% RSLogix 500 project sdss.RSS %
PROJECT "SDSS"    % processor: SLC 500, 1747-L542 %

PROGRAM FILES
  LAD 2 "MAIN"  21 rungs  %  Main Ladder Logic Program File %
  LAD 3 "TEL AZ"  17 rungs  % Telescope Azimuth Motion Control Logic File %
  LAD 5 "TEL ALT"  28 rungs  % telescope Axis Motion Control Logic File %
  LAD 7 "TEL ROT"  7 rungs  % Telescope Rotator Axis Motion Control Logic File %
  LAD 8 "INST LIFT"  106 rungs  % Instrument Lift Motion Control Logic File %
  LAD 9 "INST LATCH"  114 rungs  % Instrument Latch Control Box File %
  LAD 10 "DATA TRANS"  3 rungs  % Data Transfer subroutine for DH+ link to VME %
  LAD 11 "BRAKE STOP"  13 rungs
  LAD 12 "E-STOP SW"  19 rungs
  LAD 13 "SPEC CONT"  14 rungs  % Spectrograph Controls %
  LAD 14 "FLAT FIELD"  17 rungs  % Flat Field Lamp Controls %
  LAD 15 "FLEXANALOG"  8 rungs  % Flex I/O Analog Routines %

DATA FILES
  O0   92 elements
  I1   98 elements
  S2   164 elements
  B3   109 elements
  T4   19 elements
  C5   1 elements
  R6   1 elements
  N7   74 elements
  F8   105 elements
  B9   256 elements
  B10   48 elements
  B11   1 elements
  F12   20 elements
  B13 B13  1 elements
  N14 N14  50 elements

LADDER 2 "MAIN"    %  Main Ladder Logic Program File %
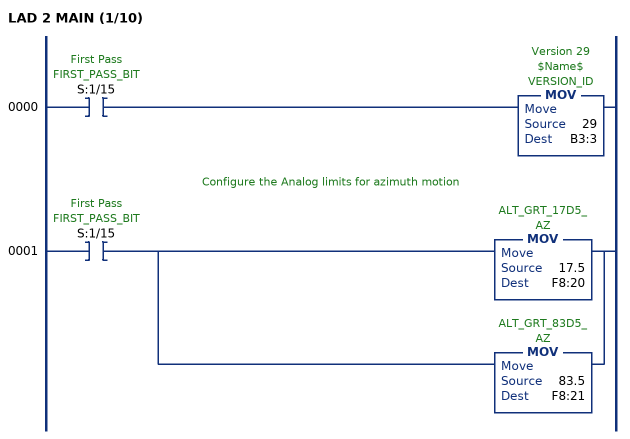
% Rung: 0 %
SOR XIC S:1/15 MOV 29 B3:3 EOR
%   S:1/15  FIRST_PASS_BIT  "First Pass" %
%   B3:3  VERSION_ID  "Version 29 $Name$" %
% Rung: 1 %
% Configure the Analog limits for azimuth motion %
SOR XIC S:1/15 BST MOV 17.5 F8:20 NXB MOV 83.5 F8:21 BND EOR
%   S:1/15  FIRST_PASS_BIT  "First Pass" %
%   F8:20  ALT_GRT_17D5_AZ %
%   F8:21  ALT_GRT_83D5_AZ %

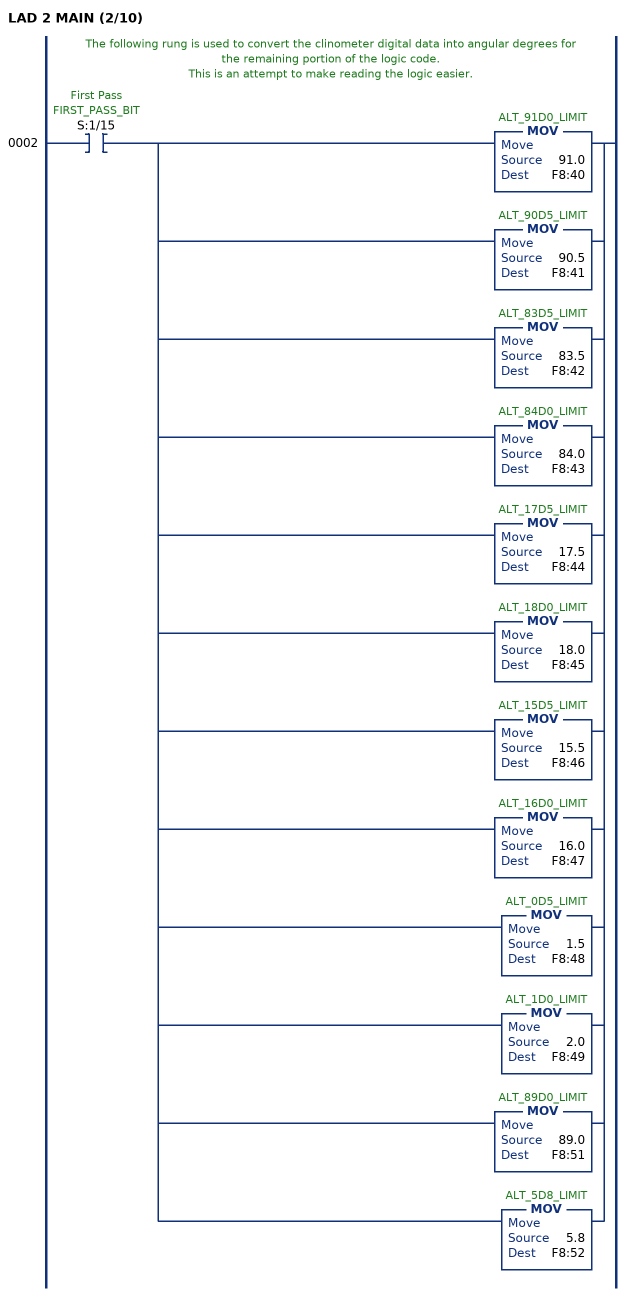
% Rung: 2 %
% The following rung is used to convert the clinometer digital data into angular degrees for the remaining portion of the logic code.
% This is an attempt to make reading the logic easier. %
SOR XIC S:1/15 BST MOV 91.0 F8:40 NXB MOV 90.5 F8:41 NXB MOV 83.5 F8:42 NXB MOV 84.0 F8:43 NXB MOV 17.5 F8:44 NXB MOV 18.0 F8:45 NXB MOV 15.5 F8:46 NXB MOV 16.0 F8:47 NXB MOV 1.5 F8:48 NXB MOV 2.0 F8:49 NXB MOV 89.0 F8:51 NXB MOV 5.8 F8:52 BND EOR
%   S:1/15  FIRST_PASS_BIT  "First Pass" %
%   F8:40  ALT_91D0_LIMIT %
%   F8:41  ALT_90D5_LIMIT %
%   F8:42  ALT_83D5_LIMIT %
%   F8:43  ALT_84D0_LIMIT %
%   F8:44  ALT_17D5_LIMIT %
%   F8:45  ALT_18D0_LIMIT %
%   F8:46  ALT_15D5_LIMIT %
%   F8:47  ALT_16D0_LIMIT %
%   F8:48  ALT_0D5_LIMIT %
%   F8:49  ALT_1D0_LIMIT %
%   F8:51  ALT_89D0_LIMIT %
%   F8:52  ALT_5D8_LIMIT %

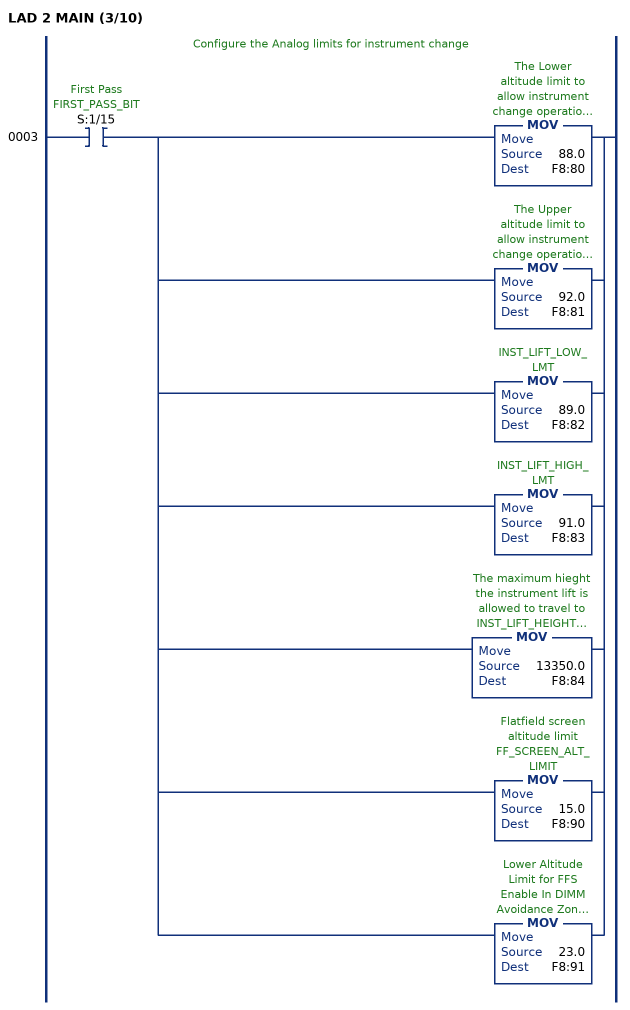
% Rung: 3 %
% Configure the Analog limits for instrument change %
SOR XIC S:1/15 BST MOV 88.0 F8:80 NXB MOV 92.0 F8:81 NXB MOV 89.0 F8:82 NXB MOV 91.0 F8:83 NXB MOV 13350.0 F8:84 NXB BST MOV 15.0 F8:90 NXB MOV 23.0 F8:91 BND BND EOR
%   S:1/15  FIRST_PASS_BIT  "First Pass" %
%   F8:80  INST_CHG_LOW_LMT  "The Lower altitude limit to allow instrument change operations" %
%   F8:81  INST_CHG_HIGH_LMT  "The Upper altitude limit to allow instrument change operations" %
%   F8:82  INST_LIFT_LOW_LMT %
%   F8:83  INST_LIFT_HIGH_LMT %
%   F8:84  INST_LIFT_HEIGHT_MAX  "The maximum hieght the instrument lift is allowed to travel to" %
%   F8:90  FF_SCREEN_ALT_LIMIT  "Flatfield screen altitude limit" %
%   F8:91  FFS_DIMM_ALT_LIM  "Lower Altitude Limit for FFS Enable In DIMM Avoidance Zone" %

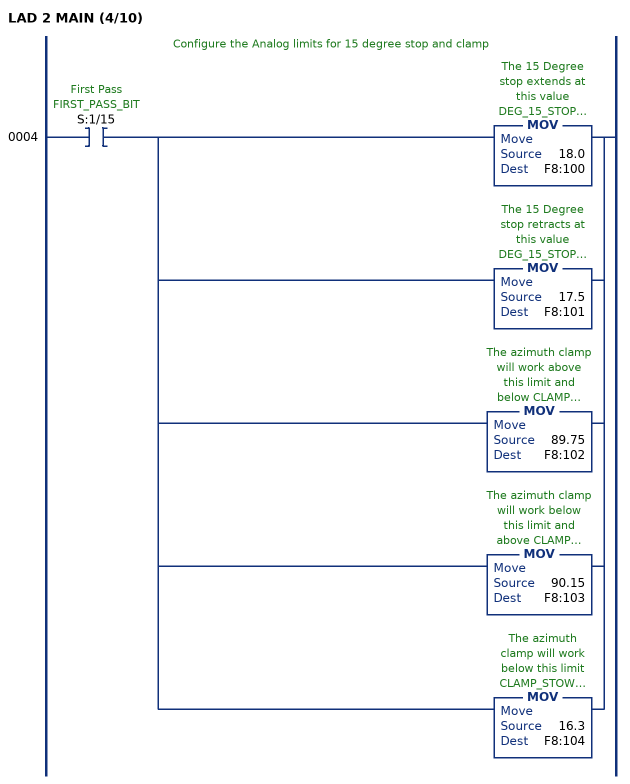
% Rung: 4 %
% Configure the Analog limits for 15 degree stop and clamp %
SOR XIC S:1/15 BST MOV 18.0 F8:100 NXB MOV 17.5 F8:101 NXB MOV 89.75 F8:102 NXB MOV 90.15 F8:103 NXB MOV 16.3 F8:104 BND EOR
%   S:1/15  FIRST_PASS_BIT  "First Pass" %
%   F8:100  DEG_15_STOP_EXT_LMT  "The 15 Degree stop extends at this value" %
%   F8:101  DEG_15_STOP_RET_LMT  "The 15 Degree stop retracts at this value" %
%   F8:102  CLAMP_LOW_LIMIT  "The azimuth clamp will work above this limit and below CLAMP_HIGH_LIMIT" %
%   F8:103  CLAMP_HIGH_LIMIT  "The azimuth clamp will work below this limit and above CLAMP_LOW_LIMIT" %
%   F8:104  CLAMP_STOW_LIMIT  "The azimuth clamp will work below this limit" %

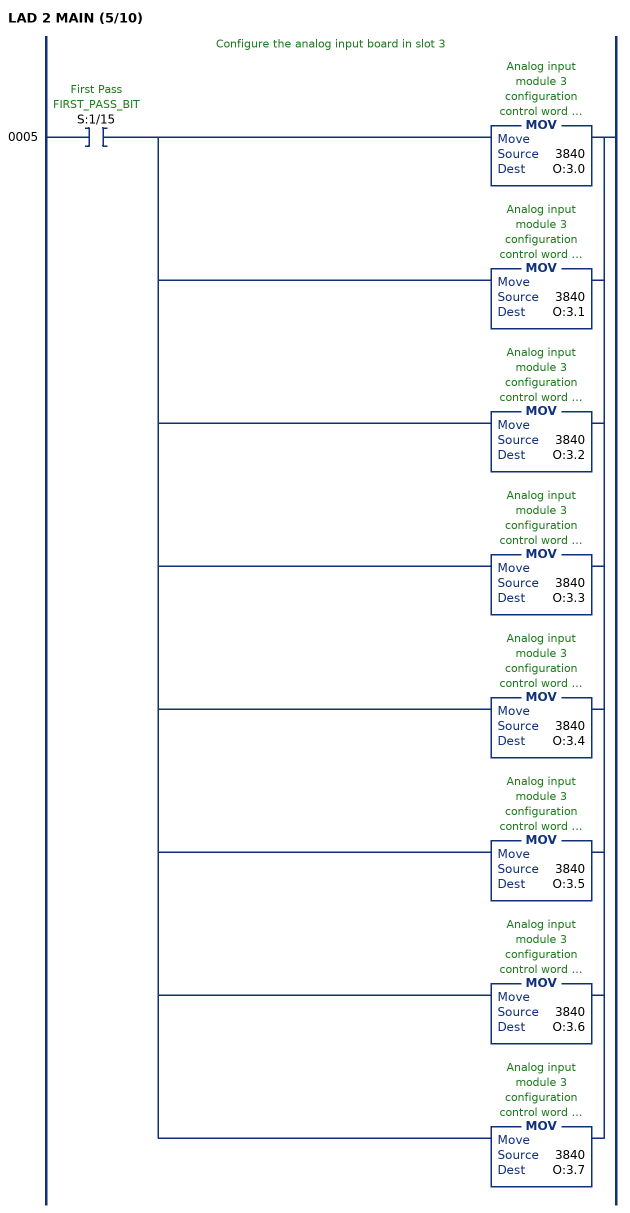
% Rung: 5 %
% Configure the analog input board in slot 3 %
SOR XIC S:1/15 BST MOV 3840 O:3.0 NXB MOV 3840 O:3.1 NXB MOV 3840 O:3.2 NXB MOV 3840 O:3.3 NXB MOV 3840 O:3.4 NXB MOV 3840 O:3.5 NXB MOV 3840 O:3.6 NXB MOV 3840 O:3.7 BND EOR
%   S:1/15  FIRST_PASS_BIT  "First Pass" %
%   O:3.0  AZ_1_VOLTAGE_CONFIG  "Analog input module 3 configuration control word 0" %
%   O:3.1  AZ_1_CURRENT_CONFIG  "Analog input module 3 configuration control word 1" %
%   O:3.2  AZ_2_VOLTAGE_CONFIG  "Analog input module 3 configuration control word 2" %
%   O:3.3  AZ_2_CURRENT_CONFIG  "Analog input module 3 configuration control word 3" %
%   O:3.4  ALT_1_VOLTAGE_CONFIG  "Analog input module 3 configuration control word 4" %
%   O:3.5  ALT_1_CURRENT_CONFIG  "Analog input module 3 configuration control word 5" %
%   O:3.6  ALT_2_VOLTAGE_CONFIG  "Analog input module 3 configuration control word 6" %
%   O:3.7  ALT_2_CURRENT_CONFIG  "Analog input module 3 configuration control word 7" %

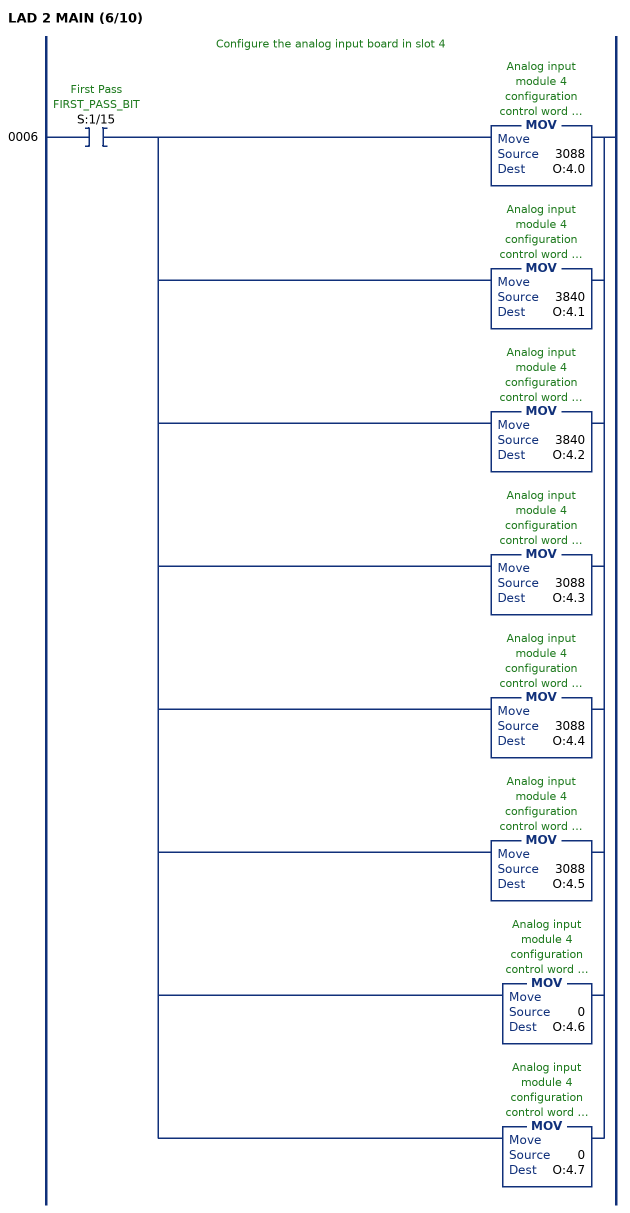
% Rung: 6 %
% Configure the analog input board in slot 4 %
SOR XIC S:1/15 BST MOV 3088 O:4.0 NXB MOV 3840 O:4.1 NXB MOV 3840 O:4.2 NXB MOV 3088 O:4.3 NXB MOV 3088 O:4.4 NXB MOV 3088 O:4.5 NXB MOV 0 O:4.6 NXB MOV 0 O:4.7 BND EOR
%   S:1/15  FIRST_PASS_BIT  "First Pass" %
%   O:4.0  ALT_POSITION_CONFIG  "Analog input module 4 configuration control word 0" %
%   O:4.1  ROT_1_VOLTAGE_CONFIG  "Analog input module 4 configuration control word 1" %
%   O:4.2  ROT_1_CURRENT_CONFIG  "Analog input module 4 configuration control word 2" %
%   O:4.3  UMBILICAL_DIST_CONFI  "Analog input module 4 configuration control word 3" %
%   O:4.4  INST_LIFT_FORCE_CONF  "Analog input module 4 configuration control word 4" %
%   O:4.5  INST_LIFT_DIST_CONFI  "Analog input module 4 configuration control word 5" %
%   O:4.6  I_4_ANALOG_6_CONFIG  "Analog input module 4 configuration control word 6" %
%   O:4.7  I_4_ANALOG_7_CONFIG  "Analog input module 4 configuration control word 7" %

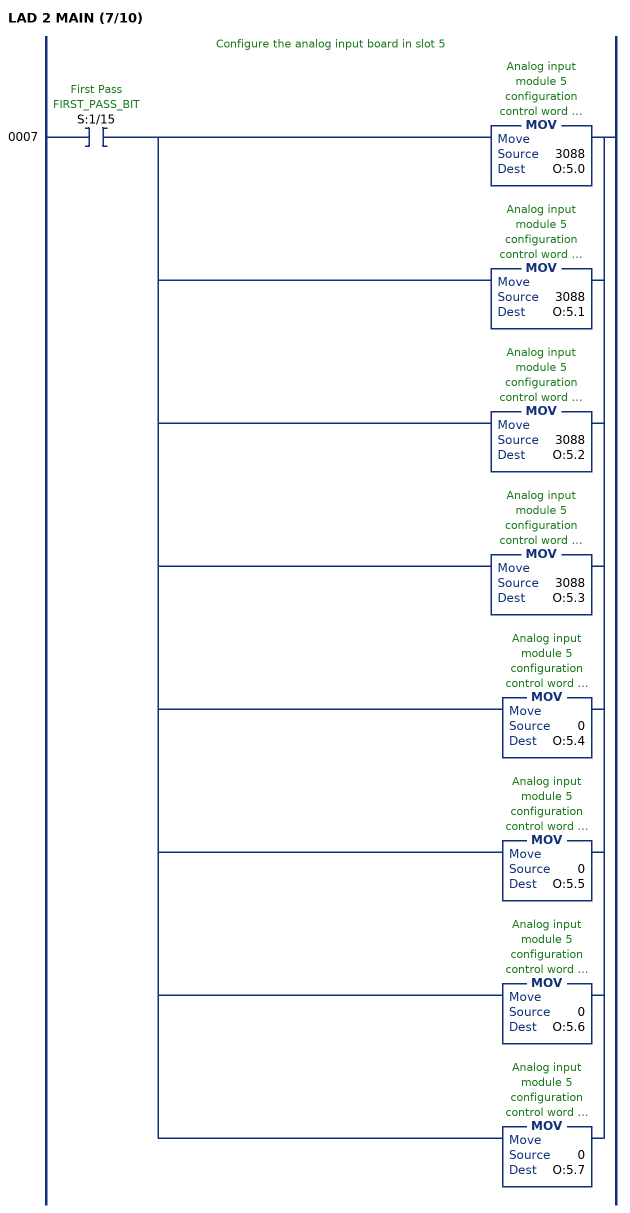
% Rung: 7 %
% Configure the analog input board in slot 5 %
SOR XIC S:1/15 BST MOV 3088 O:5.0 NXB MOV 3088 O:5.1 NXB MOV 3088 O:5.2 NXB MOV 3088 O:5.3 NXB MOV 0 O:5.4 NXB MOV 0 O:5.5 NXB MOV 0 O:5.6 NXB MOV 0 O:5.7 BND EOR
%   S:1/15  FIRST_PASS_BIT  "First Pass" %
%   O:5.0  CNTRWHT_1_POS_CONFIG  "Analog input module 5 configuration control word 0" %
%   O:5.1  CNTRWHT_2_POS_CONFIG  "Analog input module 5 configuration control word 1" %
%   O:5.2  CNTRWHT_3_POS_CONFIG  "Analog input module 5 configuration control word 2" %
%   O:5.3  CNTRWHT_4_POS_CONFIG  "Analog input module 5 configuration control word 3" %
%   O:5.4  I_5_ANALOG_4_CONFIG  "Analog input module 5 configuration control word 4" %
%   O:5.5  I_5_ANALOG_5_CONFIG  "Analog input module 5 configuration control word 5" %
%   O:5.6  I_5_ANALOG_6_CONFIG  "Analog input module 5 configuration control word 6" %
%   O:5.7  I_5_ANALOG_7_CONFIG  "Analog input module 5 configuration control word 7" %

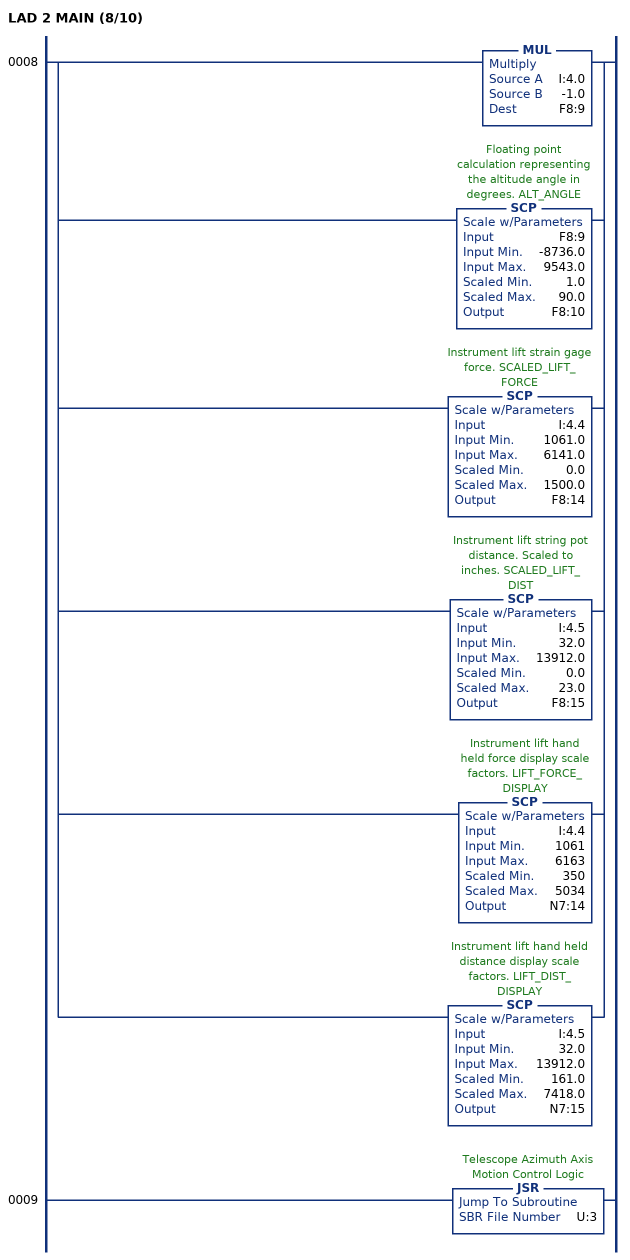
% Rung: 8 %
SOR BST MUL I:4.0 -1.0 F8:9 NXB SCP F8:9 -8736.0 9543.0 1.0 90.0 F8:10 NXB SCP I:4.4 1061.0 6141.0 0.0 1500.0 F8:14 NXB SCP I:4.5 32.0 13912.0 0.0 23.0 F8:15 NXB SCP I:4.4 1061 6163 350 5034 N7:14 NXB SCP I:4.5 32.0 13912.0 161.0 7418.0 N7:15 BND EOR
%   I:4.0  ALT_POSITION  "Altitude clinometer raw position value." %
%   F8:10  ALT_ANGLE  "Floating point calculation representing the altitude angle in degrees." %
%   I:4.4  INST_LIFT_FORCE  "Instrument lift strain gauge value." %
%   F8:14  SCALED_LIFT_FORCE  "Instrument lift strain gage force." %
%   I:4.5  INST_LIFT_DIST  "Instrument lift string pot distance value. Scale = .001,per count." 0" %
%   F8:15  SCALED_LIFT_DIST  "Instrument lift string pot distance. Scaled to inches." %
%   N7:14  LIFT_FORCE_DISPLAY  "Instrument lift hand held force display scale factors." %
%   N7:15  LIFT_DIST_DISPLAY  "Instrument lift hand held distance display scale factors." %
% Rung: 9 %
SOR JSR U:3 EOR
%   U:3  "Telescope Azimuth Axis Motion Control Logic" %

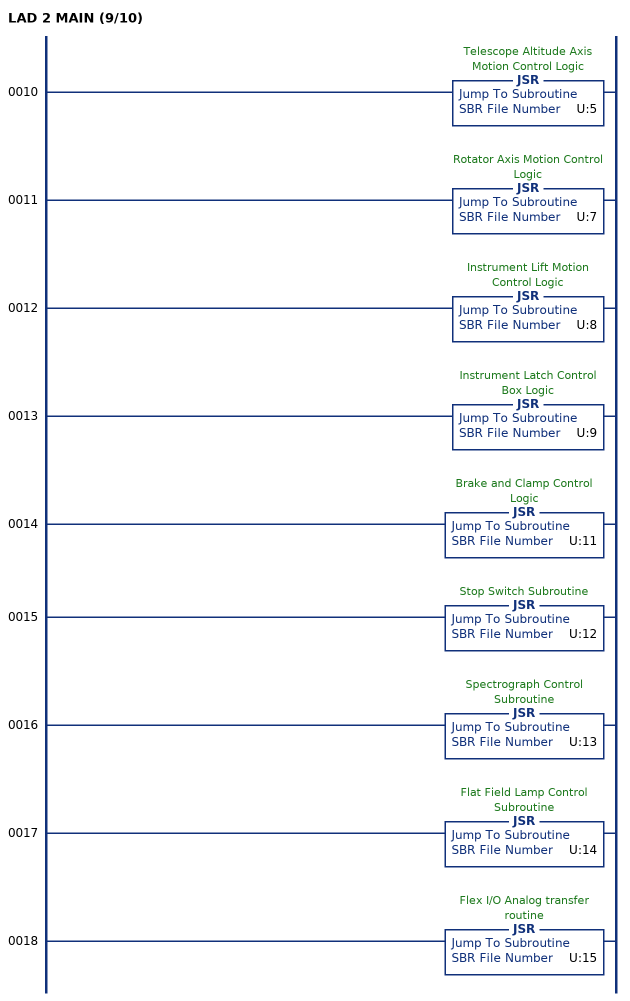
% Rung: 10 %
SOR JSR U:5 EOR
%   U:5  "Telescope Altitude Axis Motion Control Logic" %
% Rung: 11 %
SOR JSR U:7 EOR
%   U:7  "Rotator Axis Motion Control Logic" %
% Rung: 12 %
SOR JSR U:8 EOR
%   U:8  "Instrument Lift Motion Control Logic" %
% Rung: 13 %
SOR JSR U:9 EOR
%   U:9  "Instrument Latch Control Box Logic" %
% Rung: 14 %
SOR JSR U:11 EOR
%   U:11  "Brake and Clamp Control Logic" %
% Rung: 15 %
SOR JSR U:12 EOR
%   U:12  "Stop Switch Subroutine" %
% Rung: 16 %
SOR JSR U:13 EOR
%   U:13  "Spectrograph Control Subroutine" %
% Rung: 17 %
SOR JSR U:14 EOR
%   U:14  "Flat Field Lamp Control Subroutine" %
% Rung: 18 %
SOR JSR U:15 EOR
%   U:15  "Flex I/O Analog transfer routine" %

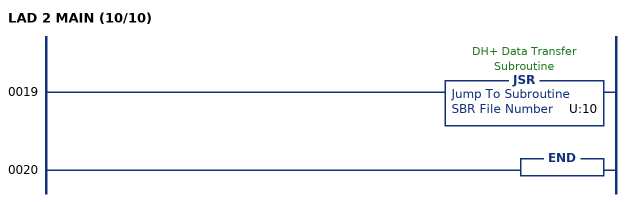
% Rung: 19 %
SOR JSR U:10 EOR
%   U:10  "DH+ Data Transfer Subroutine" %
% Rung: 20 %
SOR END EOR

LADDER 3 "TEL AZ"    % Telescope Azimuth Motion Control Logic File %
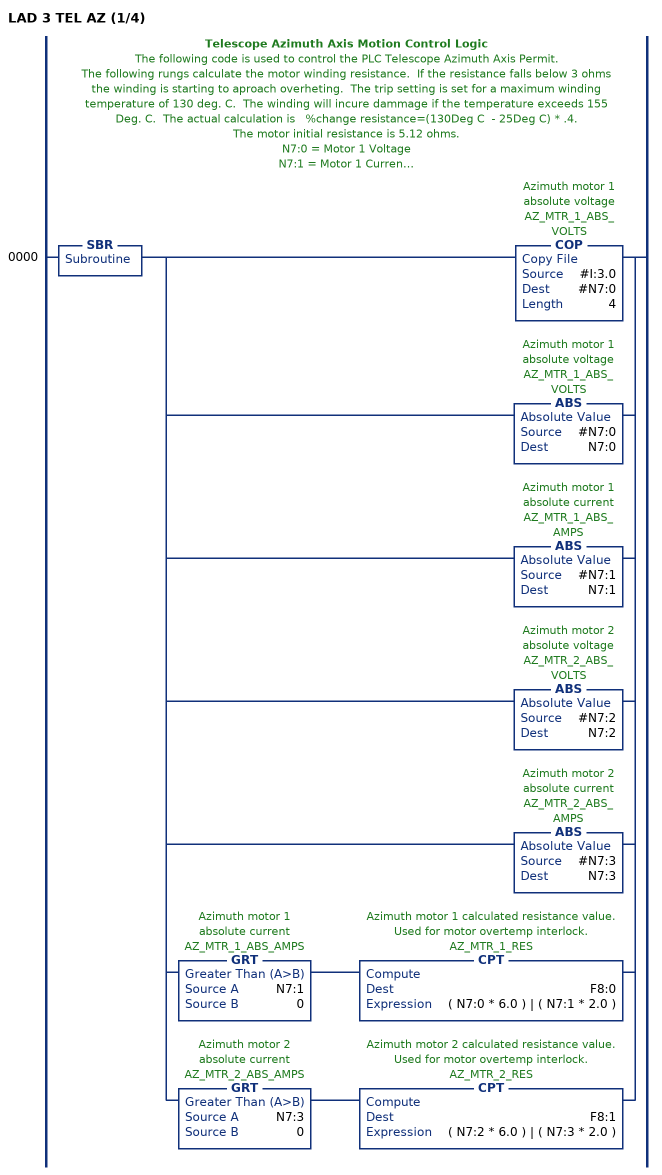
% Rung: 0 %
% TITLE: Telescope Azimuth Axis Motion Control Logic %
% The following code is used to control the PLC Telescope Azimuth Axis Permit.
% 
% 
% The following rungs calculate the motor winding resistance.  If the resistance falls below 3 ohms the winding is starting to aproach overheting.  The trip setting is set for a maximum winding temperature of 130 deg. C.  The winding will incure dammage if the temperature exceeds 155 Deg. C.  The actual calculation is   %change resistance=(130Deg C  - 25Deg C) * .4.
% 
% The motor initial resistance is 5.12 ohms.
% 
% 
% N7:0 = Motor 1 Voltage
% N7:1 = Motor 1 Current
% N7:2 = Motor 2 Voltage
% N7:3 = Motor 2 Current
% 
% If the voltage and current are not above 500 counts, then the resistance calculation is considdered invalid and an output permit is provided. %
SOR SBR BST COP #I:3.0 #N7:0 4 NXB ABS #N7:0 N7:0 NXB ABS #N7:1 N7:1 NXB ABS #N7:2 N7:2 NXB ABS #N7:3 N7:3 NXB GRT N7:1 0 CPT F8:0 " ( N7:0 * 6.0 ) | ( N7:1 * 2.0 ) " NXB GRT N7:3 0 CPT F8:1 " ( N7:2 * 6.0 ) | ( N7:3 * 2.0 ) " BND EOR
%   I:3.0  AZ_1_VOLTAGE  "Azimuth motor 1 voltage." %
%   N7:0  AZ_MTR_1_ABS_VOLTS  "Azimuth motor 1 absolute voltage" %
%   N7:1  AZ_MTR_1_ABS_AMPS  "Azimuth motor 1 absolute current" %
%   N7:2  AZ_MTR_2_ABS_VOLTS  "Azimuth motor 2 absolute voltage" %
%   N7:3  AZ_MTR_2_ABS_AMPS  "Azimuth motor 2 absolute current" %
%   F8:0  AZ_MTR_1_RES  "Azimuth motor 1 calculated resistance value. Used for motor overtemp interlock." %
%   F8:1  AZ_MTR_2_RES  "Azimuth motor 2 calculated resistance value. Used for motor overtemp interlock." %

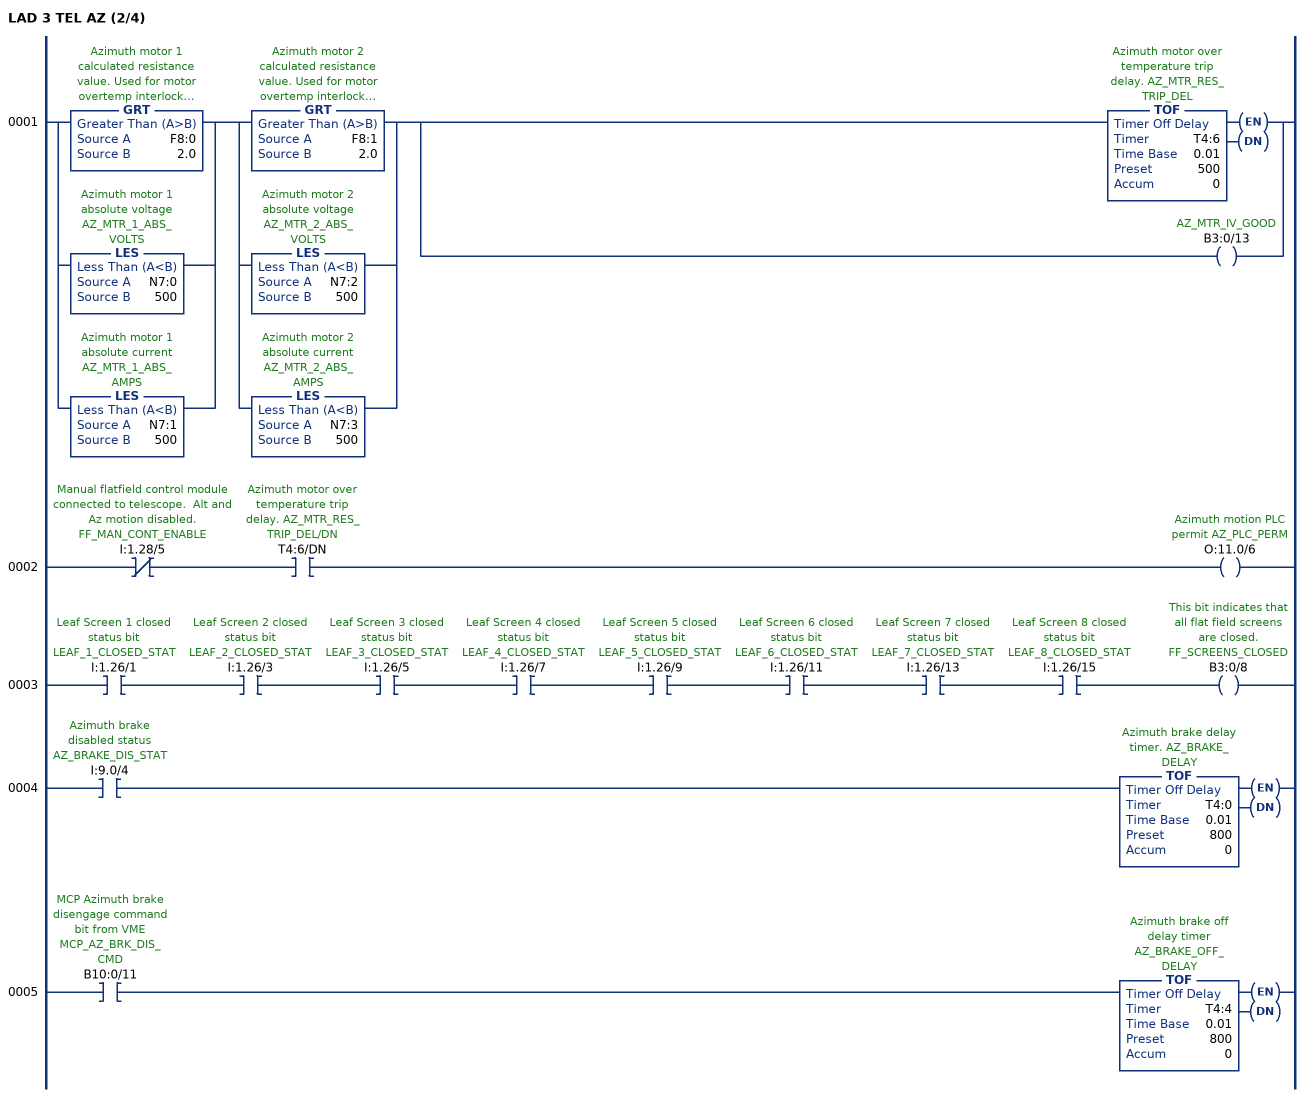
% Rung: 1 %
SOR BST GRT F8:0 2.0 NXB LES N7:0 500 NXB LES N7:1 500 BND BST GRT F8:1 2.0 NXB LES N7:2 500 NXB LES N7:3 500 BND BST TOF T4:6 0.01 500 0 NXB OTE B3:0/13 BND EOR
%   F8:0  AZ_MTR_1_RES  "Azimuth motor 1 calculated resistance value. Used for motor overtemp interlock." %
%   N7:0  AZ_MTR_1_ABS_VOLTS  "Azimuth motor 1 absolute voltage" %
%   N7:1  AZ_MTR_1_ABS_AMPS  "Azimuth motor 1 absolute current" %
%   F8:1  AZ_MTR_2_RES  "Azimuth motor 2 calculated resistance value. Used for motor overtemp interlock." %
%   N7:2  AZ_MTR_2_ABS_VOLTS  "Azimuth motor 2 absolute voltage" %
%   N7:3  AZ_MTR_2_ABS_AMPS  "Azimuth motor 2 absolute current" %
%   T4:6  AZ_MTR_RES_TRIP_DEL  "Azimuth motor over temperature trip delay." %
%   B3:0/13  AZ_MTR_IV_GOOD %
% Rung: 2 %
SOR XIO I:1.28/5 XIC T4:6/DN OTE O:11.0/6 EOR
%   I:1.28/5  FF_MAN_CONT_ENABLE  "Manual flatfield control module connected to telescope.  Alt and Az motion disabled." %
%   T4:6  AZ_MTR_RES_TRIP_DEL  "Azimuth motor over temperature trip delay." %
%   O:11.0/6  AZ_PLC_PERM  "Azimuth motion PLC permit" %
% Rung: 3 %
SOR XIC I:1.26/1 XIC I:1.26/3 XIC I:1.26/5 XIC I:1.26/7 XIC I:1.26/9 XIC I:1.26/11 XIC I:1.26/13 XIC I:1.26/15 OTE B3:0/8 EOR
%   I:1.26/1  LEAF_1_CLOSED_STAT  "Leaf Screen 1 closed status bit" %
%   I:1.26/3  LEAF_2_CLOSED_STAT  "Leaf Screen 2 closed status bit" %
%   I:1.26/5  LEAF_3_CLOSED_STAT  "Leaf Screen 3 closed status bit" %
%   I:1.26/7  LEAF_4_CLOSED_STAT  "Leaf Screen 4 closed status bit" %
%   I:1.26/9  LEAF_5_CLOSED_STAT  "Leaf Screen 5 closed status bit" %
%   I:1.26/11  LEAF_6_CLOSED_STAT  "Leaf Screen 6 closed status bit" %
%   I:1.26/13  LEAF_7_CLOSED_STAT  "Leaf Screen 7 closed status bit" %
%   I:1.26/15  LEAF_8_CLOSED_STAT  "Leaf Screen 8 closed status bit" %
%   B3:0/8  FF_SCREENS_CLOSED  "This bit indicates that all flat field screens are closed." %
% Rung: 4 %
SOR XIC I:9.0/4 TOF T4:0 0.01 800 0 EOR
%   I:9.0/4  AZ_BRAKE_DIS_STAT  "Azimuth brake disabled status" %
%   T4:0  AZ_BRAKE_DELAY  "Azimuth brake delay timer." %
% Rung: 5 %
SOR XIC B10:0/11 TOF T4:4 0.01 800 0 EOR
%   B10:0/11  MCP_AZ_BRK_DIS_CMD  "MCP Azimuth brake disengage command bit from VME" %
%   T4:4  AZ_BRAKE_OFF_DELAY  "Azimuth brake off delay timer" %

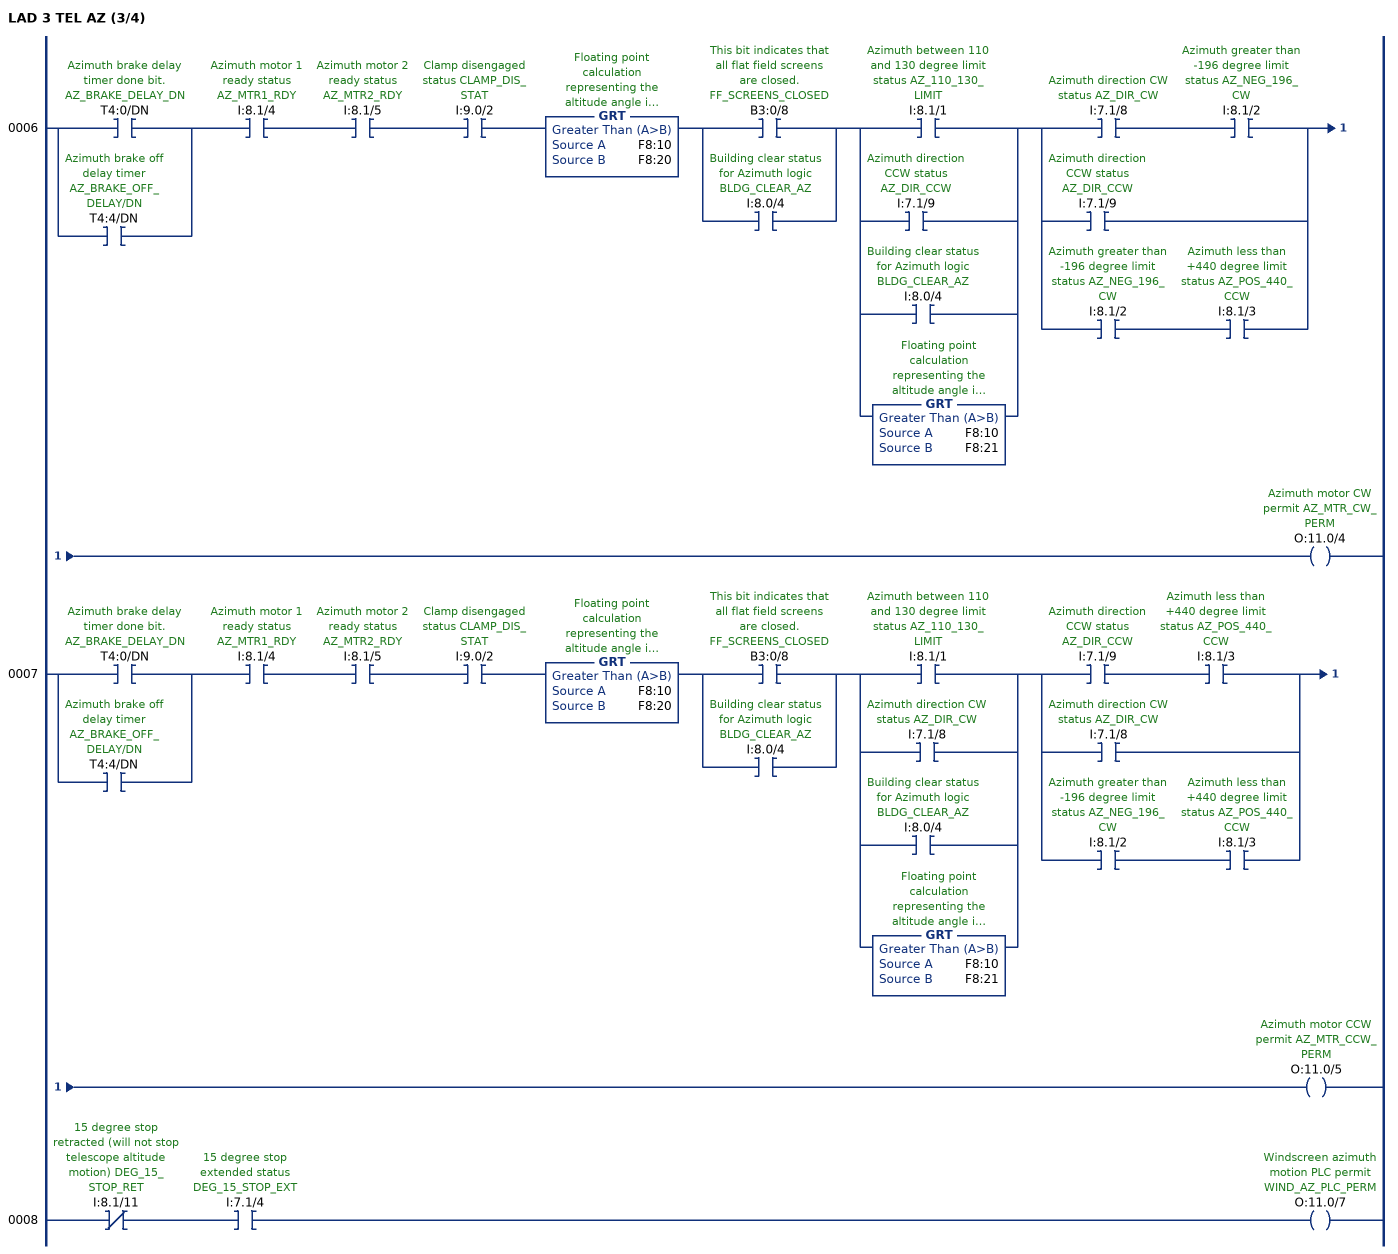
% Rung: 6 %
SOR BST XIC T4:0/DN NXB XIC T4:4/DN BND XIC I:8.1/4 XIC I:8.1/5 XIC I:9.0/2 GRT F8:10 F8:20 BST XIC B3:0/8 NXB XIC I:8.0/4 BND BST XIC I:8.1/1 NXB XIC I:7.1/9 NXB XIC I:8.0/4 NXB GRT F8:10 F8:21 BND BST XIC I:7.1/8 XIC I:8.1/2 NXB XIC I:7.1/9 NXB XIC I:8.1/2 XIC I:8.1/3 BND OTE O:11.0/4 EOR
%   T4:0/DN  AZ_BRAKE_DELAY_DN  "Azimuth brake delay timer done bit." %
%   T4:4  AZ_BRAKE_OFF_DELAY  "Azimuth brake off delay timer" %
%   I:8.1/4  AZ_MTR1_RDY  "Azimuth motor 1 ready status" %
%   I:8.1/5  AZ_MTR2_RDY  "Azimuth motor 2 ready status" %
%   I:9.0/2  CLAMP_DIS_STAT  "Clamp disengaged status" %
%   F8:10  ALT_ANGLE  "Floating point calculation representing the altitude angle in degrees." %
%   F8:20  ALT_GRT_17D5_AZ %
%   B3:0/8  FF_SCREENS_CLOSED  "This bit indicates that all flat field screens are closed." %
%   I:8.0/4  BLDG_CLEAR_AZ  "Building clear status for Azimuth logic" %
%   I:8.1/1  AZ_110_130_LIMIT  "Azimuth between 110 and 130 degree limit status" %
%   I:7.1/9  AZ_DIR_CCW  "Azimuth direction CCW status" %
%   F8:21  ALT_GRT_83D5_AZ %
%   I:7.1/8  AZ_DIR_CW  "Azimuth direction CW status" %
%   I:8.1/2  AZ_NEG_196_CW  "Azimuth greater than -196 degree limit status" %
%   I:8.1/3  AZ_POS_440_CCW  "Azimuth less than +440 degree limit status" %
%   O:11.0/4  AZ_MTR_CW_PERM  "Azimuth motor CW permit" %
% Rung: 7 %
SOR BST XIC T4:0/DN NXB XIC T4:4/DN BND XIC I:8.1/4 XIC I:8.1/5 XIC I:9.0/2 GRT F8:10 F8:20 BST XIC B3:0/8 NXB XIC I:8.0/4 BND BST XIC I:8.1/1 NXB XIC I:7.1/8 NXB XIC I:8.0/4 NXB GRT F8:10 F8:21 BND BST XIC I:7.1/9 XIC I:8.1/3 NXB XIC I:7.1/8 NXB XIC I:8.1/2 XIC I:8.1/3 BND OTE O:11.0/5 EOR
%   T4:0/DN  AZ_BRAKE_DELAY_DN  "Azimuth brake delay timer done bit." %
%   T4:4  AZ_BRAKE_OFF_DELAY  "Azimuth brake off delay timer" %
%   I:8.1/4  AZ_MTR1_RDY  "Azimuth motor 1 ready status" %
%   I:8.1/5  AZ_MTR2_RDY  "Azimuth motor 2 ready status" %
%   I:9.0/2  CLAMP_DIS_STAT  "Clamp disengaged status" %
%   F8:10  ALT_ANGLE  "Floating point calculation representing the altitude angle in degrees." %
%   F8:20  ALT_GRT_17D5_AZ %
%   B3:0/8  FF_SCREENS_CLOSED  "This bit indicates that all flat field screens are closed." %
%   I:8.0/4  BLDG_CLEAR_AZ  "Building clear status for Azimuth logic" %
%   I:8.1/1  AZ_110_130_LIMIT  "Azimuth between 110 and 130 degree limit status" %
%   I:7.1/8  AZ_DIR_CW  "Azimuth direction CW status" %
%   F8:21  ALT_GRT_83D5_AZ %
%   I:7.1/9  AZ_DIR_CCW  "Azimuth direction CCW status" %
%   I:8.1/3  AZ_POS_440_CCW  "Azimuth less than +440 degree limit status" %
%   I:8.1/2  AZ_NEG_196_CW  "Azimuth greater than -196 degree limit status" %
%   O:11.0/5  AZ_MTR_CCW_PERM  "Azimuth motor CCW permit" %
% Rung: 8 %
SOR XIO I:8.1/11 XIC I:7.1/4 OTE O:11.0/7 EOR
%   I:8.1/11  DEG_15_STOP_RET  "15 degree stop retracted (will not stop telescope altitude motion)" %
%   I:7.1/4  DEG_15_STOP_EXT  "15 degree stop extended status" %
%   O:11.0/7  WIND_AZ_PLC_PERM  "Windscreen azimuth motion PLC permit" %

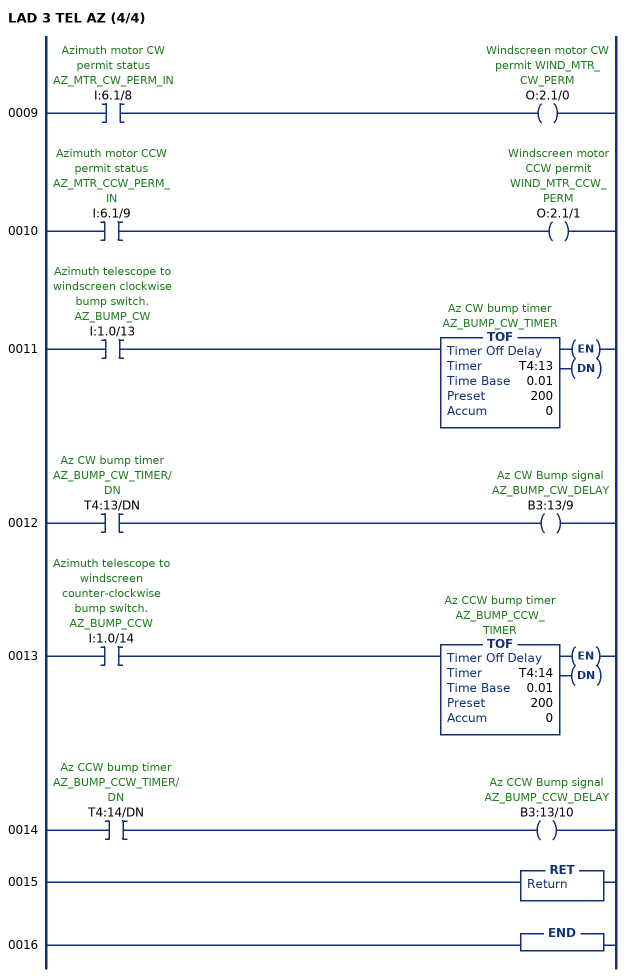
% Rung: 9 %
SOR XIC I:6.1/8 OTE O:2.1/0 EOR
%   I:6.1/8  AZ_MTR_CW_PERM_IN  "Azimuth motor CW permit status" %
%   O:2.1/0  WIND_MTR_CW_PERM  "Windscreen motor CW permit" %
% Rung: 10 %
SOR XIC I:6.1/9 OTE O:2.1/1 EOR
%   I:6.1/9  AZ_MTR_CCW_PERM_IN  "Azimuth motor CCW permit status" %
%   O:2.1/1  WIND_MTR_CCW_PERM  "Windscreen motor CCW permit" %
% Rung: 11 %
SOR XIC I:1.0/13 TOF T4:13 0.01 200 0 EOR
%   I:1.0/13  AZ_BUMP_CW  "Azimuth telescope to windscreen clockwise bump switch." %
%   T4:13  AZ_BUMP_CW_TIMER  "Az CW bump timer" %
% Rung: 12 %
SOR XIC T4:13/DN OTE B3:13/9 EOR
%   T4:13  AZ_BUMP_CW_TIMER  "Az CW bump timer" %
%   B3:13/9  AZ_BUMP_CW_DELAY  "Az CW Bump signal" %
% Rung: 13 %
SOR XIC I:1.0/14 TOF T4:14 0.01 200 0 EOR
%   I:1.0/14  AZ_BUMP_CCW  "Azimuth telescope to windscreen counter-clockwise bump switch." %
%   T4:14  AZ_BUMP_CCW_TIMER  "Az CCW bump timer" %
% Rung: 14 %
SOR XIC T4:14/DN OTE B3:13/10 EOR
%   T4:14  AZ_BUMP_CCW_TIMER  "Az CCW bump timer" %
%   B3:13/10  AZ_BUMP_CCW_DELAY  "Az CCW Bump signal" %
% Rung: 15 %
SOR RET EOR
% Rung: 16 %
SOR END EOR

LADDER 5 "TEL ALT"    % telescope Axis Motion Control Logic File %
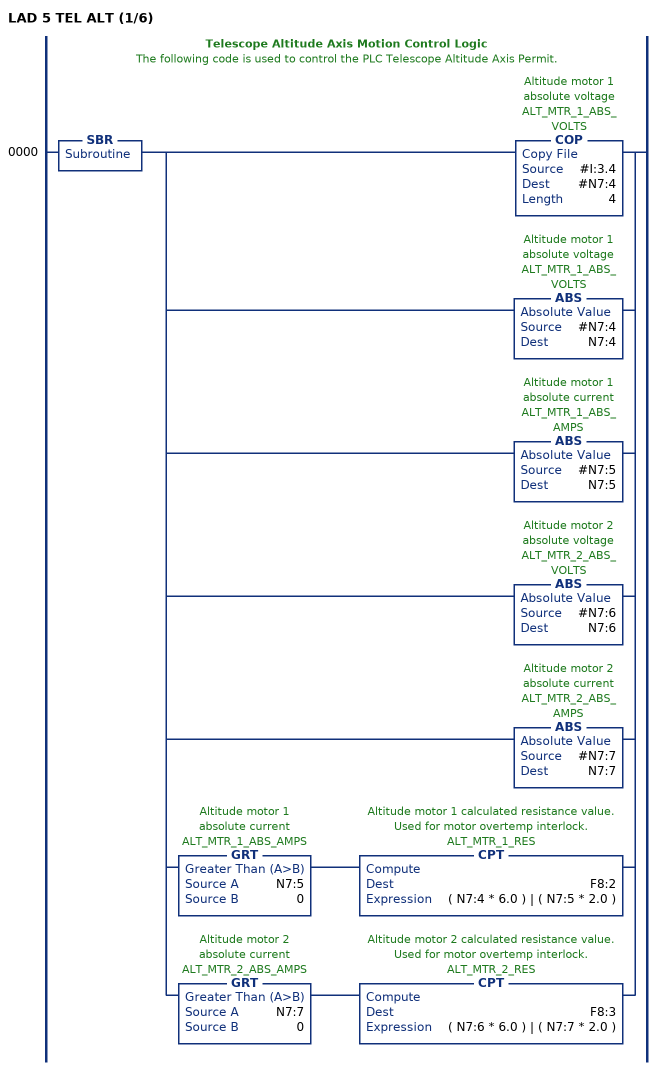
% Rung: 0 %
% TITLE: Telescope Altitude Axis Motion Control Logic %
% The following code is used to control the PLC Telescope Altitude Axis Permit. %
SOR SBR BST COP #I:3.4 #N7:4 4 NXB ABS #N7:4 N7:4 NXB ABS #N7:5 N7:5 NXB ABS #N7:6 N7:6 NXB ABS #N7:7 N7:7 NXB GRT N7:5 0 CPT F8:2 " ( N7:4 * 6.0 ) | ( N7:5 * 2.0 ) " NXB GRT N7:7 0 CPT F8:3 " ( N7:6 * 6.0 ) | ( N7:7 * 2.0 ) " BND EOR
%   I:3.4  ALT_1_VOLTAGE  "Altitude motor 1 voltage." %
%   N7:4  ALT_MTR_1_ABS_VOLTS  "Altitude motor 1 absolute voltage" %
%   N7:5  ALT_MTR_1_ABS_AMPS  "Altitude motor 1 absolute current" %
%   N7:6  ALT_MTR_2_ABS_VOLTS  "Altitude motor 2 absolute voltage" %
%   N7:7  ALT_MTR_2_ABS_AMPS  "Altitude motor 2 absolute current" %
%   F8:2  ALT_MTR_1_RES  "Altitude motor 1 calculated resistance value. Used for motor overtemp interlock." %
%   F8:3  ALT_MTR_2_RES  "Altitude motor 2 calculated resistance value. Used for motor overtemp interlock." %

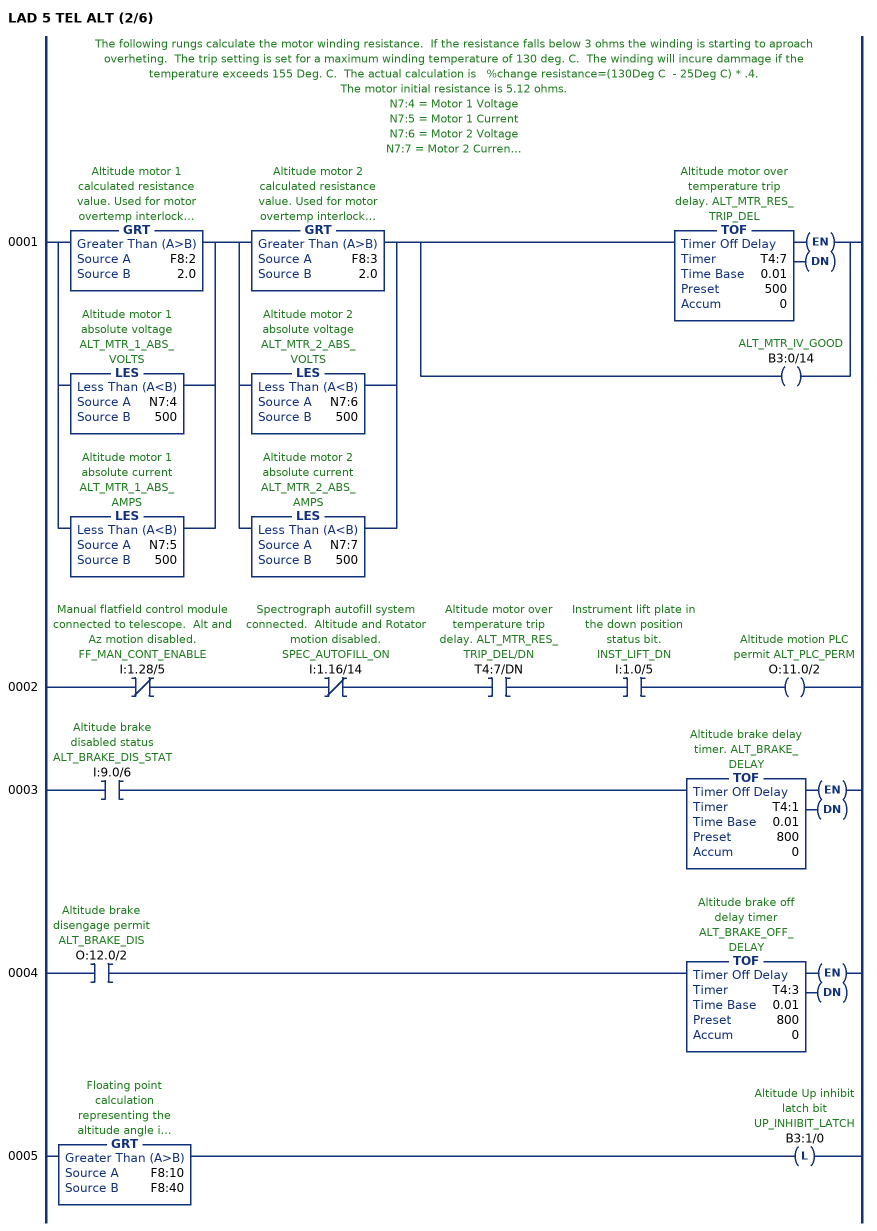
% Rung: 1 %
% The following rungs calculate the motor winding resistance.  If the resistance falls below 3 ohms the winding is starting to aproach overheting.  The trip setting is set for a maximum winding temperature of 130 deg. C.  The winding will incure dammage if the temperature exceeds 155 Deg. C.  The actual calculation is   %change resistance=(130Deg C  - 25Deg C) * .4.
% 
% The motor initial resistance is 5.12 ohms.
% 
% 
% 
% N7:4 = Motor 1 Voltage
% N7:5 = Motor 1 Current
% N7:6 = Motor 2 Voltage
% N7:7 = Motor 2 Current
% 
% If the voltage and current are not above 500 counts, then the resistance calculation is considdered invalid and an output permit is provided. %
SOR BST GRT F8:2 2.0 NXB LES N7:4 500 NXB LES N7:5 500 BND BST GRT F8:3 2.0 NXB LES N7:6 500 NXB LES N7:7 500 BND BST TOF T4:7 0.01 500 0 NXB OTE B3:0/14 BND EOR
%   F8:2  ALT_MTR_1_RES  "Altitude motor 1 calculated resistance value. Used for motor overtemp interlock." %
%   N7:4  ALT_MTR_1_ABS_VOLTS  "Altitude motor 1 absolute voltage" %
%   N7:5  ALT_MTR_1_ABS_AMPS  "Altitude motor 1 absolute current" %
%   F8:3  ALT_MTR_2_RES  "Altitude motor 2 calculated resistance value. Used for motor overtemp interlock." %
%   N7:6  ALT_MTR_2_ABS_VOLTS  "Altitude motor 2 absolute voltage" %
%   N7:7  ALT_MTR_2_ABS_AMPS  "Altitude motor 2 absolute current" %
%   T4:7  ALT_MTR_RES_TRIP_DEL  "Altitude motor over temperature trip delay." %
%   B3:0/14  ALT_MTR_IV_GOOD %
% Rung: 2 %
SOR XIO I:1.28/5 XIO I:1.16/14 XIC T4:7/DN XIC I:1.0/5 OTE O:11.0/2 EOR
%   I:1.28/5  FF_MAN_CONT_ENABLE  "Manual flatfield control module connected to telescope.  Alt and Az motion disabled." %
%   I:1.16/14  SPEC_AUTOFILL_ON  "Spectrograph autofill system connected.  Altitude and Rotator motion disabled." %
%   T4:7  ALT_MTR_RES_TRIP_DEL  "Altitude motor over temperature trip delay." %
%   I:1.0/5  INST_LIFT_DN  "Instrument lift plate in the down position status bit." %
%   O:11.0/2  ALT_PLC_PERM  "Altitude motion PLC permit" %
% Rung: 3 %
SOR XIC I:9.0/6 TOF T4:1 0.01 800 0 EOR
%   I:9.0/6  ALT_BRAKE_DIS_STAT  "Altitude brake disabled status" %
%   T4:1  ALT_BRAKE_DELAY  "Altitude brake delay timer." %
% Rung: 4 %
SOR XIC O:12.0/2 TOF T4:3 0.01 800 0 EOR
%   O:12.0/2  ALT_BRAKE_DIS  "Altitude brake disengage permit" %
%   T4:3  ALT_BRAKE_OFF_DELAY  "Altitude brake off delay timer" %
% Rung: 5 %
SOR GRT F8:10 F8:40 OTL B3:1/0 EOR
%   F8:10  ALT_ANGLE  "Floating point calculation representing the altitude angle in degrees." %
%   F8:40  ALT_91D0_LIMIT %
%   B3:1/0  UP_INHIBIT_LATCH  "Altitude Up inhibit latch bit" %

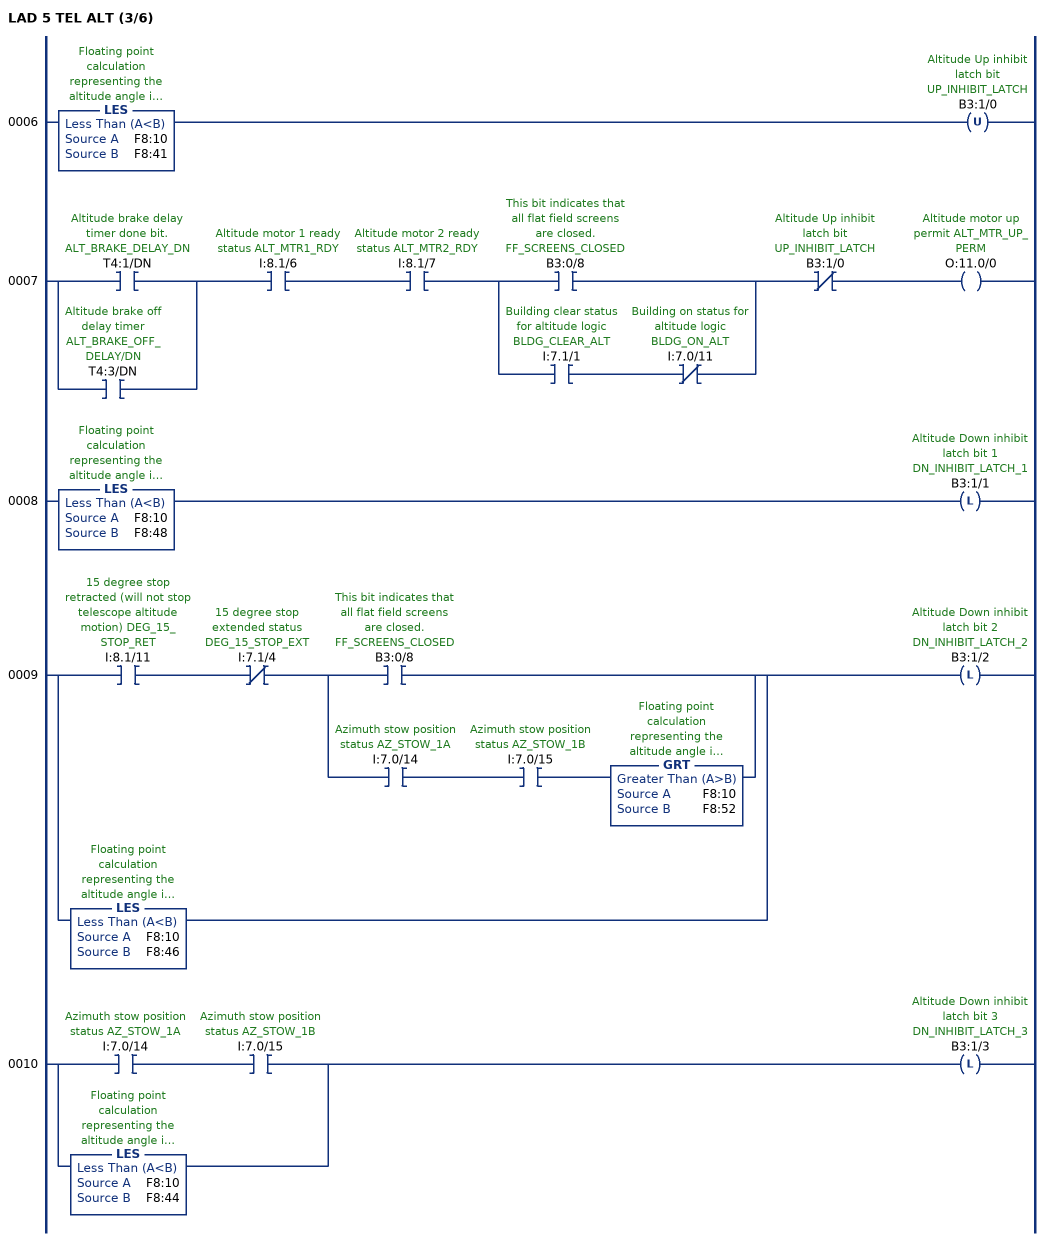
% Rung: 6 %
SOR LES F8:10 F8:41 OTU B3:1/0 EOR
%   F8:10  ALT_ANGLE  "Floating point calculation representing the altitude angle in degrees." %
%   F8:41  ALT_90D5_LIMIT %
%   B3:1/0  UP_INHIBIT_LATCH  "Altitude Up inhibit latch bit" %
% Rung: 7 %
SOR BST XIC T4:1/DN NXB XIC T4:3/DN BND XIC I:8.1/6 XIC I:8.1/7 BST XIC B3:0/8 NXB XIC I:7.1/1 XIO I:7.0/11 BND XIO B3:1/0 OTE O:11.0/0 EOR
%   T4:1/DN  ALT_BRAKE_DELAY_DN  "Altitude brake delay timer done bit." %
%   T4:3  ALT_BRAKE_OFF_DELAY  "Altitude brake off delay timer" %
%   I:8.1/6  ALT_MTR1_RDY  "Altitude motor 1 ready status" %
%   I:8.1/7  ALT_MTR2_RDY  "Altitude motor 2 ready status" %
%   B3:0/8  FF_SCREENS_CLOSED  "This bit indicates that all flat field screens are closed." %
%   I:7.1/1  BLDG_CLEAR_ALT  "Building clear status for altitude logic" %
%   I:7.0/11  BLDG_ON_ALT  "Building on status for altitude logic" %
%   B3:1/0  UP_INHIBIT_LATCH  "Altitude Up inhibit latch bit" %
%   O:11.0/0  ALT_MTR_UP_PERM  "Altitude motor up permit" %
% Rung: 8 %
SOR LES F8:10 F8:48 OTL B3:1/1 EOR
%   F8:10  ALT_ANGLE  "Floating point calculation representing the altitude angle in degrees." %
%   F8:48  ALT_0D5_LIMIT %
%   B3:1/1  DN_INHIBIT_LATCH_1  "Altitude Down inhibit latch bit 1" %
% Rung: 9 %
SOR BST XIC I:8.1/11 XIO I:7.1/4 BST XIC B3:0/8 NXB XIC I:7.0/14 XIC I:7.0/15 GRT F8:10 F8:52 BND NXB LES F8:10 F8:46 BND OTL B3:1/2 EOR
%   I:8.1/11  DEG_15_STOP_RET  "15 degree stop retracted (will not stop telescope altitude motion)" %
%   I:7.1/4  DEG_15_STOP_EXT  "15 degree stop extended status" %
%   B3:0/8  FF_SCREENS_CLOSED  "This bit indicates that all flat field screens are closed." %
%   I:7.0/14  AZ_STOW_1A  "Azimuth stow position status" %
%   I:7.0/15  AZ_STOW_1B  "Azimuth stow position status" %
%   F8:10  ALT_ANGLE  "Floating point calculation representing the altitude angle in degrees." %
%   F8:52  ALT_5D8_LIMIT %
%   F8:46  ALT_15D5_LIMIT %
%   B3:1/2  DN_INHIBIT_LATCH_2  "Altitude Down inhibit latch bit 2" %
% Rung: 10 %
SOR BST XIC I:7.0/14 XIC I:7.0/15 NXB LES F8:10 F8:44 BND OTL B3:1/3 EOR
%   I:7.0/14  AZ_STOW_1A  "Azimuth stow position status" %
%   I:7.0/15  AZ_STOW_1B  "Azimuth stow position status" %
%   F8:10  ALT_ANGLE  "Floating point calculation representing the altitude angle in degrees." %
%   F8:44  ALT_17D5_LIMIT %
%   B3:1/3  DN_INHIBIT_LATCH_3  "Altitude Down inhibit latch bit 3" %

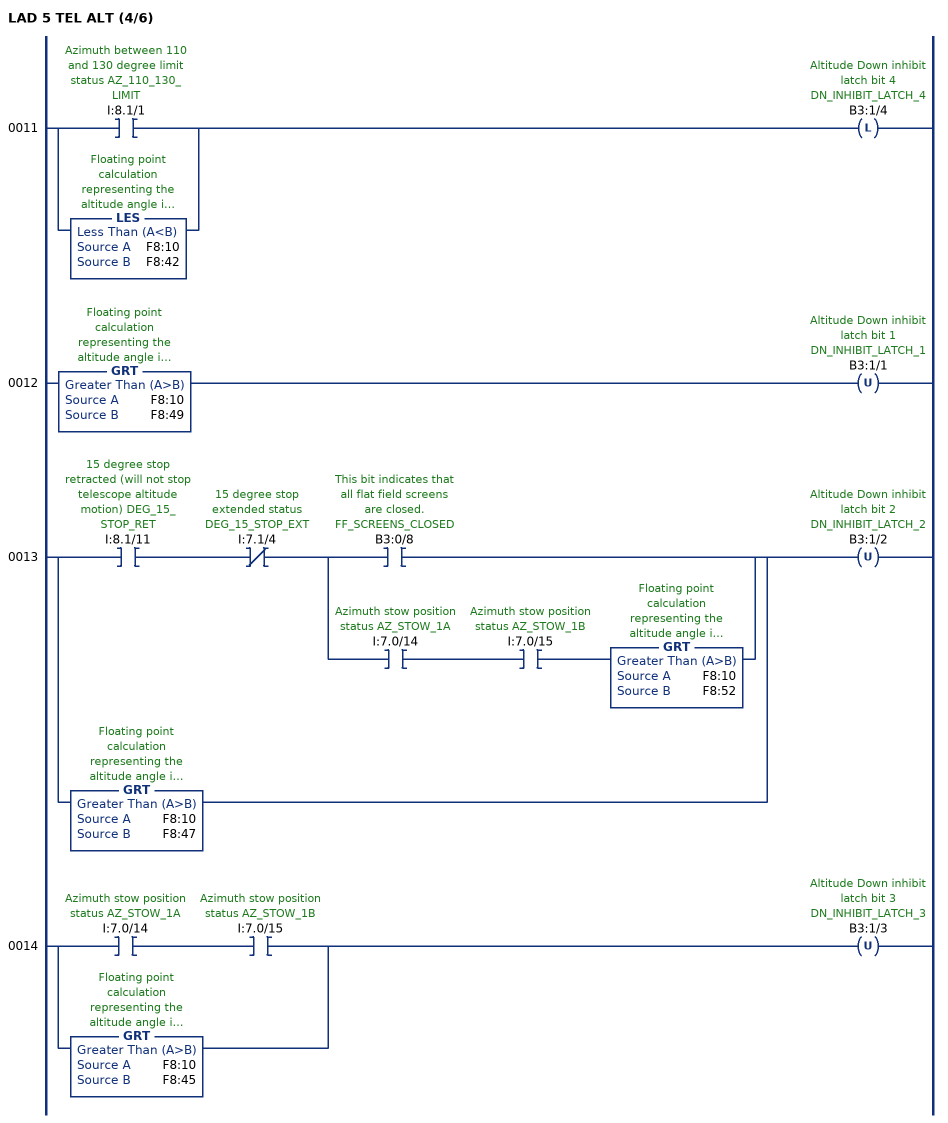
% Rung: 11 %
SOR BST XIC I:8.1/1 NXB LES F8:10 F8:42 BND OTL B3:1/4 EOR
%   I:8.1/1  AZ_110_130_LIMIT  "Azimuth between 110 and 130 degree limit status" %
%   F8:10  ALT_ANGLE  "Floating point calculation representing the altitude angle in degrees." %
%   F8:42  ALT_83D5_LIMIT %
%   B3:1/4  DN_INHIBIT_LATCH_4  "Altitude Down inhibit latch bit 4" %
% Rung: 12 %
SOR GRT F8:10 F8:49 OTU B3:1/1 EOR
%   F8:10  ALT_ANGLE  "Floating point calculation representing the altitude angle in degrees." %
%   F8:49  ALT_1D0_LIMIT %
%   B3:1/1  DN_INHIBIT_LATCH_1  "Altitude Down inhibit latch bit 1" %
% Rung: 13 %
SOR BST XIC I:8.1/11 XIO I:7.1/4 BST XIC B3:0/8 NXB XIC I:7.0/14 XIC I:7.0/15 GRT F8:10 F8:52 BND NXB GRT F8:10 F8:47 BND OTU B3:1/2 EOR
%   I:8.1/11  DEG_15_STOP_RET  "15 degree stop retracted (will not stop telescope altitude motion)" %
%   I:7.1/4  DEG_15_STOP_EXT  "15 degree stop extended status" %
%   B3:0/8  FF_SCREENS_CLOSED  "This bit indicates that all flat field screens are closed." %
%   I:7.0/14  AZ_STOW_1A  "Azimuth stow position status" %
%   I:7.0/15  AZ_STOW_1B  "Azimuth stow position status" %
%   F8:10  ALT_ANGLE  "Floating point calculation representing the altitude angle in degrees." %
%   F8:52  ALT_5D8_LIMIT %
%   F8:47  ALT_16D0_LIMIT %
%   B3:1/2  DN_INHIBIT_LATCH_2  "Altitude Down inhibit latch bit 2" %
% Rung: 14 %
SOR BST XIC I:7.0/14 XIC I:7.0/15 NXB GRT F8:10 F8:45 BND OTU B3:1/3 EOR
%   I:7.0/14  AZ_STOW_1A  "Azimuth stow position status" %
%   I:7.0/15  AZ_STOW_1B  "Azimuth stow position status" %
%   F8:10  ALT_ANGLE  "Floating point calculation representing the altitude angle in degrees." %
%   F8:45  ALT_18D0_LIMIT %
%   B3:1/3  DN_INHIBIT_LATCH_3  "Altitude Down inhibit latch bit 3" %

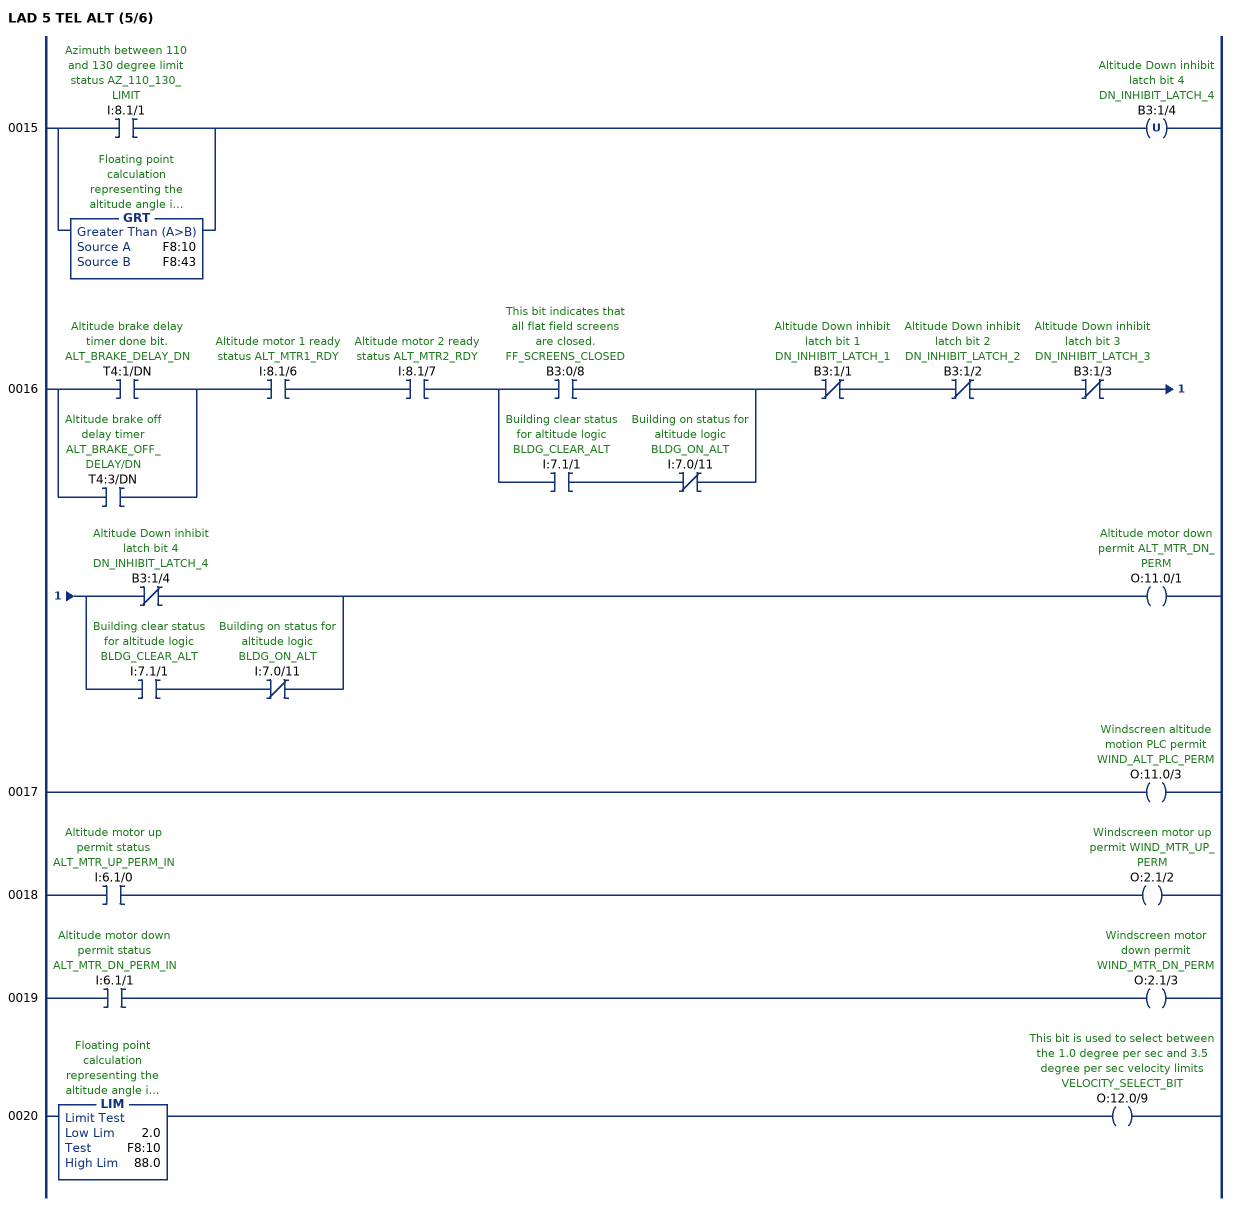
% Rung: 15 %
SOR BST XIC I:8.1/1 NXB GRT F8:10 F8:43 BND OTU B3:1/4 EOR
%   I:8.1/1  AZ_110_130_LIMIT  "Azimuth between 110 and 130 degree limit status" %
%   F8:10  ALT_ANGLE  "Floating point calculation representing the altitude angle in degrees." %
%   F8:43  ALT_84D0_LIMIT %
%   B3:1/4  DN_INHIBIT_LATCH_4  "Altitude Down inhibit latch bit 4" %
% Rung: 16 %
SOR BST XIC T4:1/DN NXB XIC T4:3/DN BND XIC I:8.1/6 XIC I:8.1/7 BST XIC B3:0/8 NXB XIC I:7.1/1 XIO I:7.0/11 BND XIO B3:1/1 XIO B3:1/2 XIO B3:1/3 BST XIO B3:1/4 NXB XIC I:7.1/1 XIO I:7.0/11 BND OTE O:11.0/1 EOR
%   T4:1/DN  ALT_BRAKE_DELAY_DN  "Altitude brake delay timer done bit." %
%   T4:3  ALT_BRAKE_OFF_DELAY  "Altitude brake off delay timer" %
%   I:8.1/6  ALT_MTR1_RDY  "Altitude motor 1 ready status" %
%   I:8.1/7  ALT_MTR2_RDY  "Altitude motor 2 ready status" %
%   B3:0/8  FF_SCREENS_CLOSED  "This bit indicates that all flat field screens are closed." %
%   I:7.1/1  BLDG_CLEAR_ALT  "Building clear status for altitude logic" %
%   I:7.0/11  BLDG_ON_ALT  "Building on status for altitude logic" %
%   B3:1/1  DN_INHIBIT_LATCH_1  "Altitude Down inhibit latch bit 1" %
%   B3:1/2  DN_INHIBIT_LATCH_2  "Altitude Down inhibit latch bit 2" %
%   B3:1/3  DN_INHIBIT_LATCH_3  "Altitude Down inhibit latch bit 3" %
%   B3:1/4  DN_INHIBIT_LATCH_4  "Altitude Down inhibit latch bit 4" %
%   O:11.0/1  ALT_MTR_DN_PERM  "Altitude motor down permit" %
% Rung: 17 %
SOR OTE O:11.0/3 EOR
%   O:11.0/3  WIND_ALT_PLC_PERM  "Windscreen altitude motion PLC permit" %
% Rung: 18 %
SOR XIC I:6.1/0 OTE O:2.1/2 EOR
%   I:6.1/0  ALT_MTR_UP_PERM_IN  "Altitude motor up permit status" %
%   O:2.1/2  WIND_MTR_UP_PERM  "Windscreen motor up permit" %
% Rung: 19 %
SOR XIC I:6.1/1 OTE O:2.1/3 EOR
%   I:6.1/1  ALT_MTR_DN_PERM_IN  "Altitude motor down permit status" %
%   O:2.1/3  WIND_MTR_DN_PERM  "Windscreen motor down permit" %
% Rung: 20 %
SOR LIM 2.0 F8:10 88.0 OTE O:12.0/9 EOR
%   F8:10  ALT_ANGLE  "Floating point calculation representing the altitude angle in degrees." %
%   O:12.0/9  VELOCITY_SELECT_BIT  "This bit is used to select between the 1.0 degree per sec and 3.5 degree per sec velocity limits" %

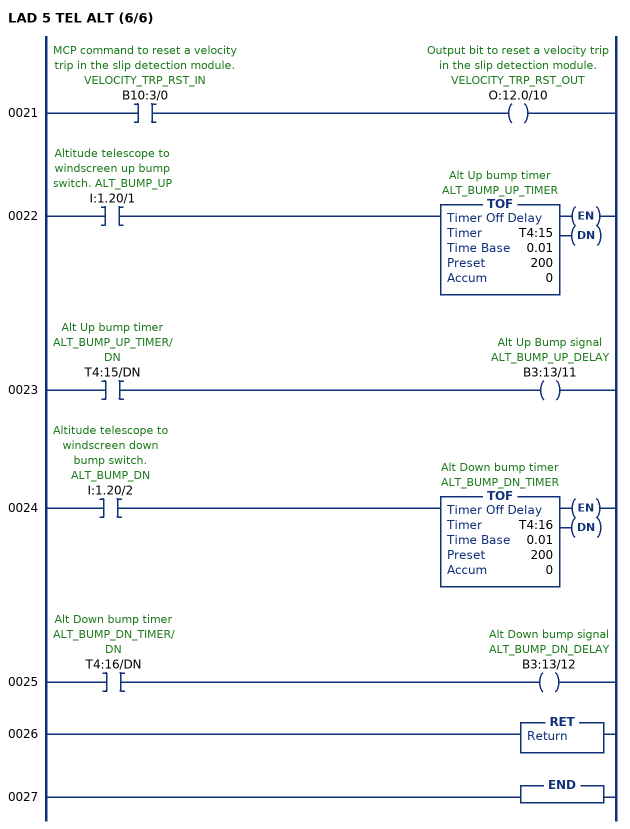
% Rung: 21 %
SOR XIC B10:3/0 OTE O:12.0/10 EOR
%   B10:3/0  VELOCITY_TRP_RST_IN  "MCP command to reset a velocity trip in the slip detection module." %
%   O:12.0/10  VELOCITY_TRP_RST_OUT  "Output bit to reset a velocity trip in the slip detection module." %
% Rung: 22 %
SOR XIC I:1.20/1 TOF T4:15 0.01 200 0 EOR
%   I:1.20/1  ALT_BUMP_UP  "Altitude telescope to windscreen up bump switch." %
%   T4:15  ALT_BUMP_UP_TIMER  "Alt Up bump timer" %
% Rung: 23 %
SOR XIC T4:15/DN OTE B3:13/11 EOR
%   T4:15  ALT_BUMP_UP_TIMER  "Alt Up bump timer" %
%   B3:13/11  ALT_BUMP_UP_DELAY  "Alt Up Bump signal" %
% Rung: 24 %
SOR XIC I:1.20/2 TOF T4:16 0.01 200 0 EOR
%   I:1.20/2  ALT_BUMP_DN  "Altitude telescope to windscreen down bump switch." %
%   T4:16  ALT_BUMP_DN_TIMER  "Alt Down bump timer" %
% Rung: 25 %
SOR XIC T4:16/DN OTE B3:13/12 EOR
%   T4:16  ALT_BUMP_DN_TIMER  "Alt Down bump timer" %
%   B3:13/12  ALT_BUMP_DN_DELAY  "Alt Down bump signal" %
% Rung: 26 %
SOR RET EOR
% Rung: 27 %
SOR END EOR

LADDER 7 "TEL ROT"    % Telescope Rotator Axis Motion Control Logic File %
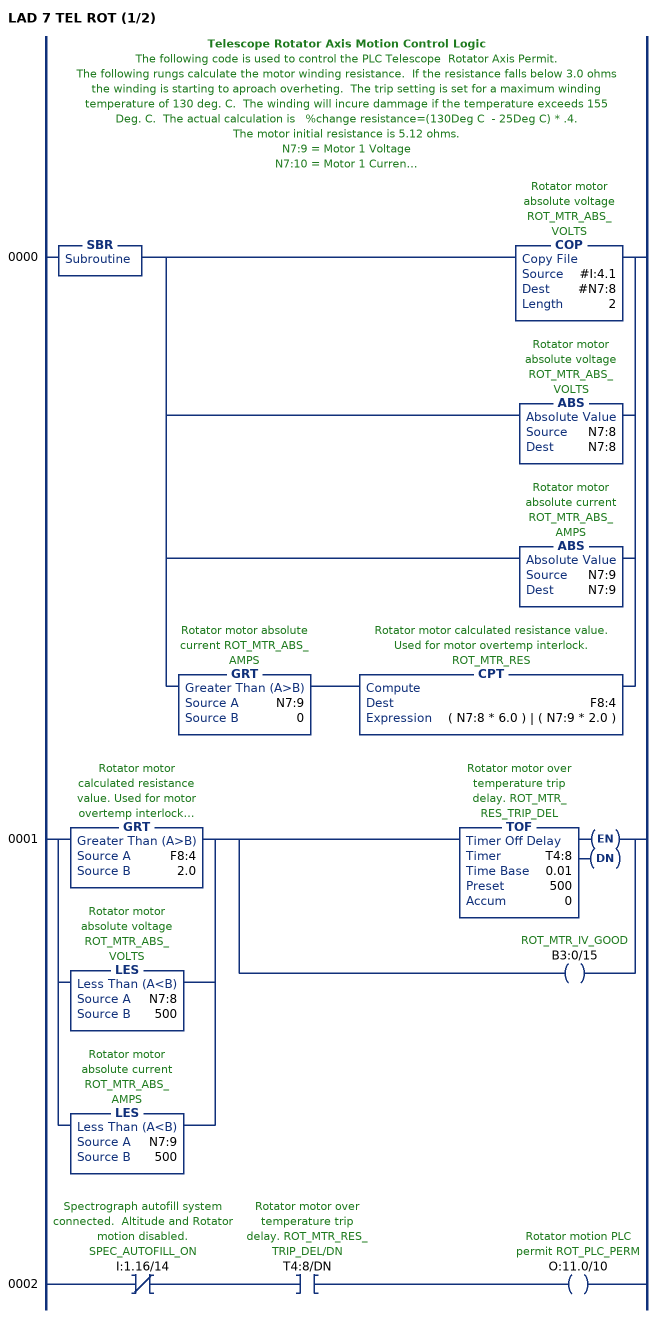
% Rung: 0 %
% TITLE: Telescope Rotator Axis Motion Control Logic %
% The following code is used to control the PLC Telescope  Rotator Axis Permit.
% 
% 
% The following rungs calculate the motor winding resistance.  If the resistance falls below 3.0 ohms the winding is starting to aproach overheting.  The trip setting is set for a maximum winding temperature of 130 deg. C.  The winding will incure dammage if the temperature exceeds 155 Deg. C.  The actual calculation is   %change resistance=(130Deg C  - 25Deg C) * .4.
% 
% The motor initial resistance is 5.12 ohms.
% 
% 
% 
% N7:9 = Motor 1 Voltage
% N7:10 = Motor 1 Current
% 
% If the voltage and current are not above 500 counts, then the resistance calculation is considdered invalid and an output permit is provided. %
SOR SBR BST COP #I:4.1 #N7:8 2 NXB ABS N7:8 N7:8 NXB ABS N7:9 N7:9 NXB GRT N7:9 0 CPT F8:4 " ( N7:8 * 6.0 ) | ( N7:9 * 2.0 ) " BND EOR
%   I:4.1  ROT_1_VOLTAGE  "Rotator motor voltage." %
%   N7:8  ROT_MTR_ABS_VOLTS  "Rotator motor absolute voltage" %
%   N7:9  ROT_MTR_ABS_AMPS  "Rotator motor absolute current" %
%   F8:4  ROT_MTR_RES  "Rotator motor calculated resistance value. Used for motor overtemp interlock." %
% Rung: 1 %
SOR BST GRT F8:4 2.0 NXB LES N7:8 500 NXB LES N7:9 500 BND BST TOF T4:8 0.01 500 0 NXB OTE B3:0/15 BND EOR
%   F8:4  ROT_MTR_RES  "Rotator motor calculated resistance value. Used for motor overtemp interlock." %
%   N7:8  ROT_MTR_ABS_VOLTS  "Rotator motor absolute voltage" %
%   N7:9  ROT_MTR_ABS_AMPS  "Rotator motor absolute current" %
%   T4:8  ROT_MTR_RES_TRIP_DEL  "Rotator motor over temperature trip delay." %
%   B3:0/15  ROT_MTR_IV_GOOD %
% Rung: 2 %
SOR XIO I:1.16/14 XIC T4:8/DN OTE O:11.0/10 EOR
%   I:1.16/14  SPEC_AUTOFILL_ON  "Spectrograph autofill system connected.  Altitude and Rotator motion disabled." %
%   T4:8  ROT_MTR_RES_TRIP_DEL  "Rotator motor over temperature trip delay." %
%   O:11.0/10  ROT_PLC_PERM  "Rotator motion PLC permit" %

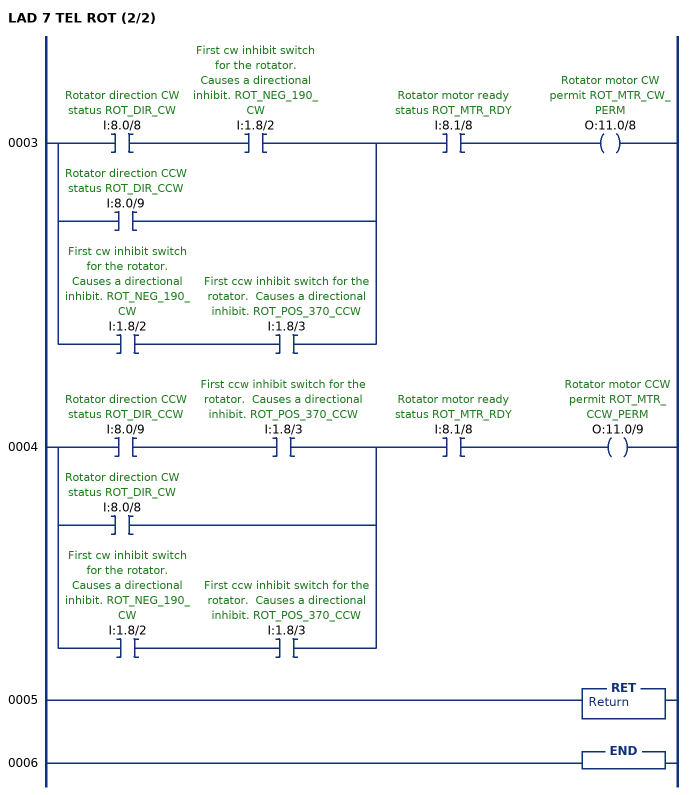
% Rung: 3 %
SOR BST XIC I:8.0/8 XIC I:1.8/2 NXB XIC I:8.0/9 NXB XIC I:1.8/2 XIC I:1.8/3 BND XIC I:8.1/8 OTE O:11.0/8 EOR
%   I:8.0/8  ROT_DIR_CW  "Rotator direction CW status" %
%   I:1.8/2  ROT_NEG_190_CW  "First cw inhibit switch for the rotator.  Causes a directional inhibit." %
%   I:8.0/9  ROT_DIR_CCW  "Rotator direction CCW status" %
%   I:1.8/3  ROT_POS_370_CCW  "First ccw inhibit switch for the rotator.  Causes a directional inhibit." %
%   I:8.1/8  ROT_MTR_RDY  "Rotator motor ready status" %
%   O:11.0/8  ROT_MTR_CW_PERM  "Rotator motor CW permit" %
% Rung: 4 %
SOR BST XIC I:8.0/9 XIC I:1.8/3 NXB XIC I:8.0/8 NXB XIC I:1.8/2 XIC I:1.8/3 BND XIC I:8.1/8 OTE O:11.0/9 EOR
%   I:8.0/9  ROT_DIR_CCW  "Rotator direction CCW status" %
%   I:1.8/3  ROT_POS_370_CCW  "First ccw inhibit switch for the rotator.  Causes a directional inhibit." %
%   I:8.0/8  ROT_DIR_CW  "Rotator direction CW status" %
%   I:1.8/2  ROT_NEG_190_CW  "First cw inhibit switch for the rotator.  Causes a directional inhibit." %
%   I:8.1/8  ROT_MTR_RDY  "Rotator motor ready status" %
%   O:11.0/9  ROT_MTR_CCW_PERM  "Rotator motor CCW permit" %
% Rung: 5 %
SOR RET EOR
% Rung: 6 %
SOR END EOR

LADDER 8 "INST LIFT"    % Instrument Lift Motion Control Logic File %
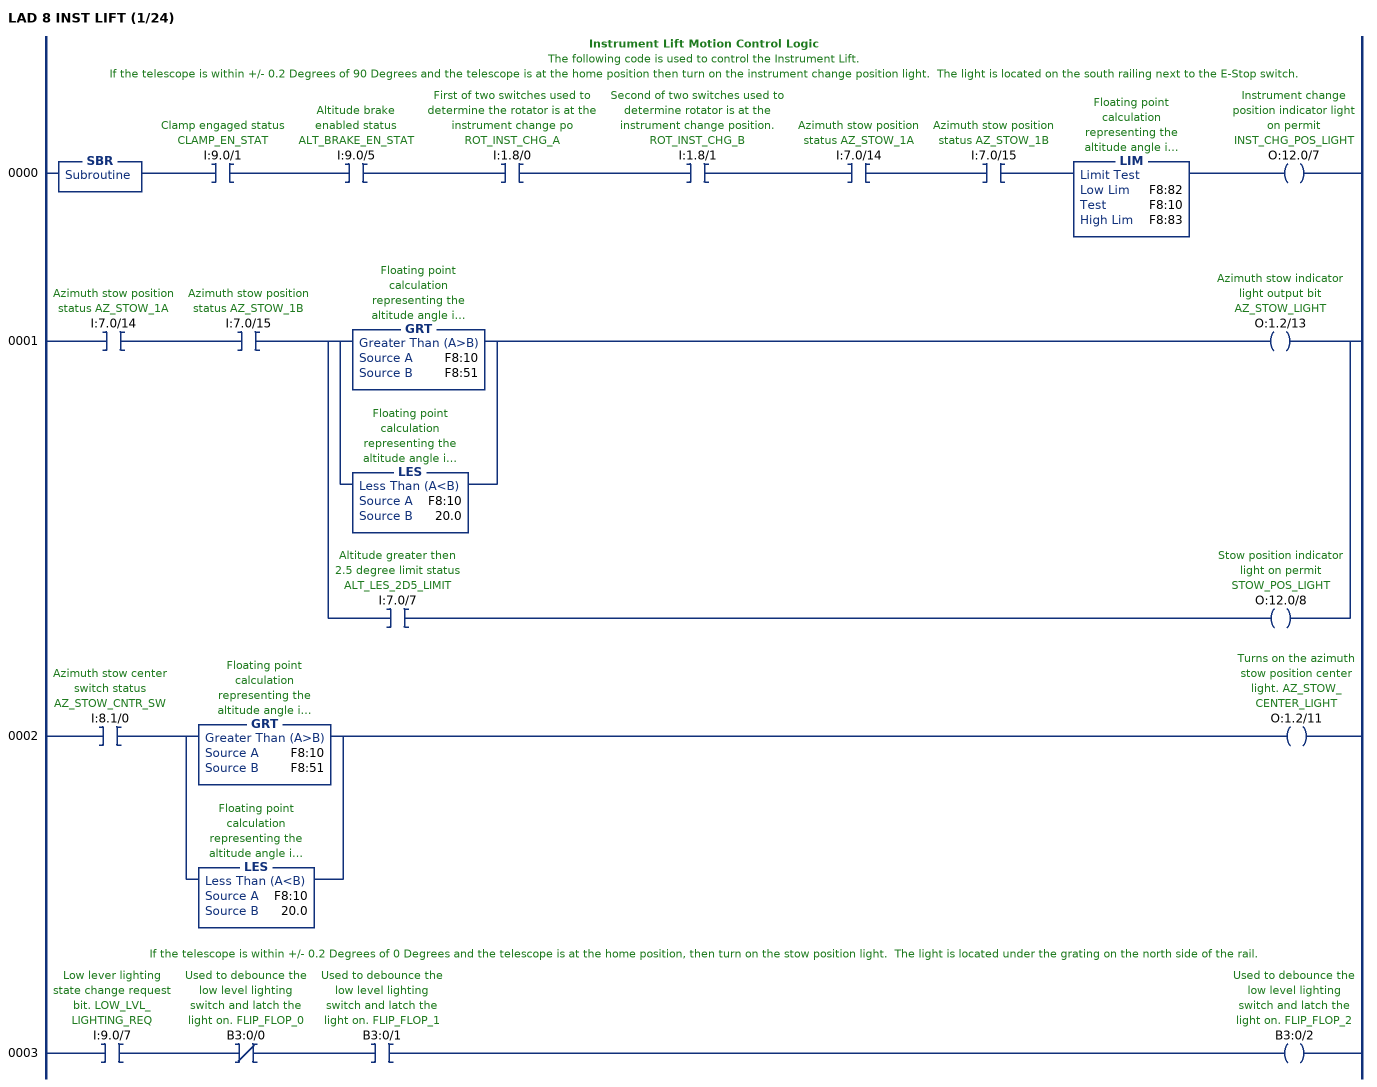
% Rung: 0 %
% TITLE: Instrument Lift Motion Control Logic %
% The following code is used to control the Instrument Lift.
% 
% If the telescope is within +/- 0.2 Degrees of 90 Degrees and the telescope is at the home position then turn on the instrument change position light.  The light is located on the south railing next to the E-Stop switch. %
SOR SBR XIC I:9.0/1 XIC I:9.0/5 XIC I:1.8/0 XIC I:1.8/1 XIC I:7.0/14 XIC I:7.0/15 LIM F8:82 F8:10 F8:83 OTE O:12.0/7 EOR
%   I:9.0/1  CLAMP_EN_STAT  "Clamp engaged status" %
%   I:9.0/5  ALT_BRAKE_EN_STAT  "Altitude brake enabled status" %
%   I:1.8/0  ROT_INST_CHG_A  "First of two switches used to determine the rotator is at the instrument change po" %
%   I:1.8/1  ROT_INST_CHG_B  "Second of two switches used to determine rotator is at the instrument change position." %
%   I:7.0/14  AZ_STOW_1A  "Azimuth stow position status" %
%   I:7.0/15  AZ_STOW_1B  "Azimuth stow position status" %
%   F8:82  INST_LIFT_LOW_LMT %
%   F8:10  ALT_ANGLE  "Floating point calculation representing the altitude angle in degrees." %
%   F8:83  INST_LIFT_HIGH_LMT %
%   O:12.0/7  INST_CHG_POS_LIGHT  "Instrument change position indicator light on permit" %
% Rung: 1 %
SOR XIC I:7.0/14 XIC I:7.0/15 BST BST GRT F8:10 F8:51 NXB LES F8:10 20.0 BND OTE O:1.2/13 NXB XIC I:7.0/7 OTE O:12.0/8 BND EOR
%   I:7.0/14  AZ_STOW_1A  "Azimuth stow position status" %
%   I:7.0/15  AZ_STOW_1B  "Azimuth stow position status" %
%   F8:10  ALT_ANGLE  "Floating point calculation representing the altitude angle in degrees." %
%   F8:51  ALT_89D0_LIMIT %
%   O:1.2/13  AZ_STOW_LIGHT  "Azimuth stow indicator light output bit" %
%   I:7.0/7  ALT_LES_2D5_LIMIT  "Altitude greater then 2.5 degree limit status" %
%   O:12.0/8  STOW_POS_LIGHT  "Stow position indicator light on permit" %
% Rung: 2 %
SOR XIC I:8.1/0 BST GRT F8:10 F8:51 NXB LES F8:10 20.0 BND OTE O:1.2/11 EOR
%   I:8.1/0  AZ_STOW_CNTR_SW  "Azimuth stow center switch status" %
%   F8:10  ALT_ANGLE  "Floating point calculation representing the altitude angle in degrees." %
%   F8:51  ALT_89D0_LIMIT %
%   O:1.2/11  AZ_STOW_CENTER_LIGHT  "Turns on the azimuth stow position center light." %
% Rung: 3 %
%  If the telescope is within +/- 0.2 Degrees of 0 Degrees and the telescope is at the home position, then turn on the stow position light.  The light is located under the grating on the north side of the rail. %
SOR XIC I:9.0/7 XIO B3:0/0 XIC B3:0/1 OTE B3:0/2 EOR
%   I:9.0/7  LOW_LVL_LIGHTING_REQ  "Low lever lighting state change request bit." %
%   B3:0/0  FLIP_FLOP_0  "Used to debounce the low level lighting switch and latch the light on." %
%   B3:0/1  FLIP_FLOP_1  "Used to debounce the low level lighting switch and latch the light on." %
%   B3:0/2  FLIP_FLOP_2  "Used to debounce the low level lighting switch and latch the light on." %

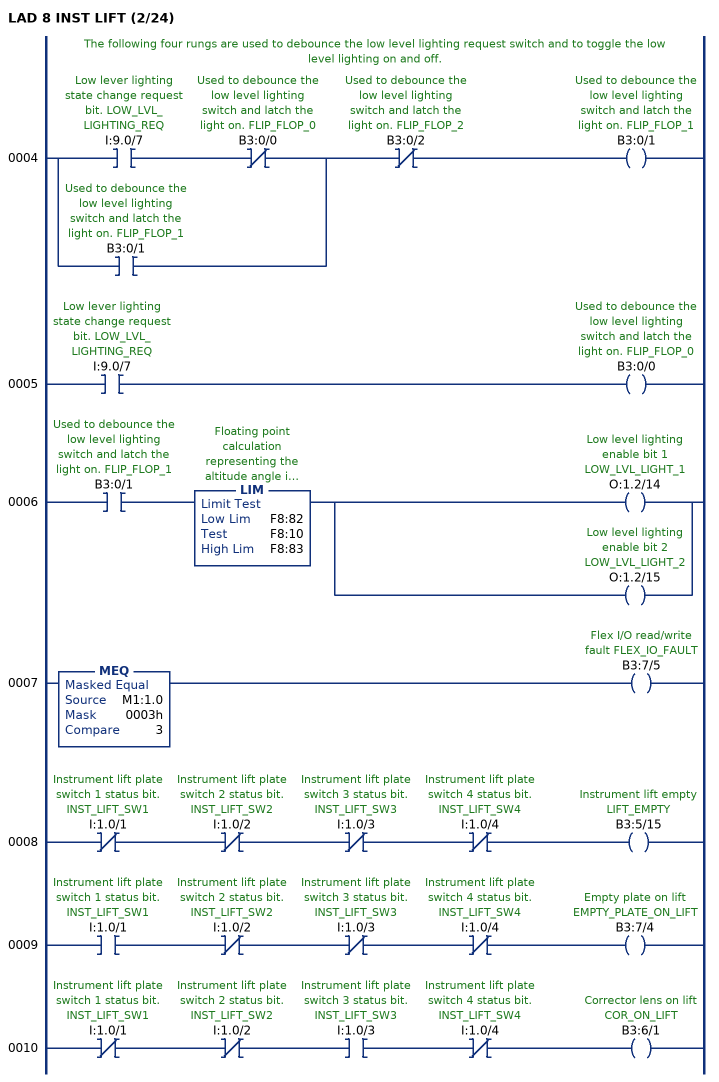
% Rung: 4 %
% The following four rungs are used to debounce the low level lighting request switch and to toggle the low level lighting on and off. %
SOR BST XIC I:9.0/7 XIO B3:0/0 NXB XIC B3:0/1 BND XIO B3:0/2 OTE B3:0/1 EOR
%   I:9.0/7  LOW_LVL_LIGHTING_REQ  "Low lever lighting state change request bit." %
%   B3:0/0  FLIP_FLOP_0  "Used to debounce the low level lighting switch and latch the light on." %
%   B3:0/1  FLIP_FLOP_1  "Used to debounce the low level lighting switch and latch the light on." %
%   B3:0/2  FLIP_FLOP_2  "Used to debounce the low level lighting switch and latch the light on." %
% Rung: 5 %
SOR XIC I:9.0/7 OTE B3:0/0 EOR
%   I:9.0/7  LOW_LVL_LIGHTING_REQ  "Low lever lighting state change request bit." %
%   B3:0/0  FLIP_FLOP_0  "Used to debounce the low level lighting switch and latch the light on." %
% Rung: 6 %
SOR XIC B3:0/1 LIM F8:82 F8:10 F8:83 BST OTE O:1.2/14 NXB OTE O:1.2/15 BND EOR
%   B3:0/1  FLIP_FLOP_1  "Used to debounce the low level lighting switch and latch the light on." %
%   F8:82  INST_LIFT_LOW_LMT %
%   F8:10  ALT_ANGLE  "Floating point calculation representing the altitude angle in degrees." %
%   F8:83  INST_LIFT_HIGH_LMT %
%   O:1.2/14  LOW_LVL_LIGHT_1  "Low level lighting enable bit 1" %
%   O:1.2/15  LOW_LVL_LIGHT_2  "Low level lighting enable bit 2" %
% Rung: 7 %
SOR MEQ M1:1.0 0003h 3 OTE B3:7/5 EOR
%   B3:7/5  FLEX_IO_FAULT  "Flex I/O read/write fault" %
% Rung: 8 %
SOR XIO I:1.0/1 XIO I:1.0/2 XIO I:1.0/3 XIO I:1.0/4 OTE B3:5/15 EOR
%   I:1.0/1  INST_LIFT_SW1  "Instrument lift plate switch 1 status bit." %
%   I:1.0/2  INST_LIFT_SW2  "Instrument lift plate switch 2 status bit." %
%   I:1.0/3  INST_LIFT_SW3  "Instrument lift plate switch 3 status bit." %
%   I:1.0/4  INST_LIFT_SW4  "Instrument lift plate switch 4 status bit." %
%   B3:5/15  LIFT_EMPTY  "Instrument lift empty" %
% Rung: 9 %
SOR XIC I:1.0/1 XIO I:1.0/2 XIO I:1.0/3 XIO I:1.0/4 OTE B3:7/4 EOR
%   I:1.0/1  INST_LIFT_SW1  "Instrument lift plate switch 1 status bit." %
%   I:1.0/2  INST_LIFT_SW2  "Instrument lift plate switch 2 status bit." %
%   I:1.0/3  INST_LIFT_SW3  "Instrument lift plate switch 3 status bit." %
%   I:1.0/4  INST_LIFT_SW4  "Instrument lift plate switch 4 status bit." %
%   B3:7/4  EMPTY_PLATE_ON_LIFT  "Empty plate on lift" %
% Rung: 10 %
SOR XIO I:1.0/1 XIO I:1.0/2 XIC I:1.0/3 XIO I:1.0/4 OTE B3:6/1 EOR
%   I:1.0/1  INST_LIFT_SW1  "Instrument lift plate switch 1 status bit." %
%   I:1.0/2  INST_LIFT_SW2  "Instrument lift plate switch 2 status bit." %
%   I:1.0/3  INST_LIFT_SW3  "Instrument lift plate switch 3 status bit." %
%   I:1.0/4  INST_LIFT_SW4  "Instrument lift plate switch 4 status bit." %
%   B3:6/1  COR_ON_LIFT  "Corrector lens on lift" %

